C07257=1094.933,100.327,-61.473,176.140,17.129,152.422
C07258=1094.927,100.078,-61.455,176.137,17.128,152.422
C07259=1094.922,99.829,-61.436,176.135,17.127,152.422
C07260=1094.916,99.579,-61.418,176.132,17.127,152.423
C07261=1094.911,99.330,-61.401,176.130,17.125,152.423
C07262=1094.905,99.081,-61.381,176.128,17.125,152.423
C07263=1094.899,98.832,-61.364,176.125,17.124,152.424
C07264=1094.893,98.582,-61.346,176.123,17.123,152.424
C07265=1094.888,98.333,-61.327,176.120,17.123,152.424
C07266=1094.882,98.083,-61.309,176.117,17.121,152.425
C07267=1094.877,97.834,-61.291,176.115,17.121,152.425
C07268=1094.870,97.585,-61.274,176.112,17.120,152.425
C07269=1094.865,97.336,-61.255,176.110,17.119,152.426
C07270=1094.859,97.086,-61.237,176.108,17.118,152.426
C07271=1094.854,96.837,-61.219,176.106,17.117,152.426
C07272=1094.848,96.587,-61.201,176.103,17.117,152.426
C07273=1094.843,96.339,-61.182,176.100,17.115,152.427
C07274=1094.836,96.063,-61.163,176.098,17.115,152.427
C07275=1094.830,95.788,-61.143,176.095,17.114,152.427
C07276=1094.824,95.513,-61.123,176.093,17.113,152.428
C07277=1094.817,95.237,-61.104,176.090,17.112,152.428
C07278=1094.812,94.988,-61.085,176.087,17.111,152.428
C07279=1094.806,94.739,-61.067,176.085,17.110,152.429
C07280=1094.801,94.490,-61.049,176.082,17.109,152.429
C07281=1094.794,94.240,-61.031,176.080,17.108,152.429
C07282=1094.790,93.991,-61.013,176.077,17.108,152.430
C07283=1094.784,93.741,-60.995,176.075,17.107,152.430
C07284=1094.778,93.492,-60.978,176.073,17.106,152.430
C07285=1094.772,93.243,-60.960,176.070,17.104,152.430
C07286=1094.767,92.993,-60.941,176.068,17.104,152.431
C07287=1094.761,92.744,-60.923,176.065,17.103,152.431
C07288=1094.756,92.495,-60.906,176.063,17.102,152.431
C07289=1094.750,92.245,-60.888,176.061,17.101,152.432
C07290=1094.744,91.996,-60.870,176.059,17.101,152.432
C07291=1094.739,91.747,-60.852,176.056,17.099,152.432
C07292=1094.733,91.497,-60.834,176.054,17.099,152.432
C07293=1094.728,91.248,-60.816,176.051,17.097,152.433
C07294=1094.722,90.999,-60.799,176.048,17.097,152.433
C07295=1094.716,90.749,-60.781,176.046,17.096,152.433
C07296=1094.711,90.500,-60.763,176.044,17.095,152.434
C07297=1094.705,90.251,-60.746,176.042,17.094,152.434
C07298=1094.699,90.002,-60.728,176.039,17.093,152.434
C07299=1094.693,89.753,-60.710,176.037,17.093,152.434
C07300=1094.688,89.504,-60.693,176.034,17.092,152.435
C07301=1094.682,89.254,-60.675,176.032,17.091,152.435
C07302=1094.676,89.005,-60.657,176.030,17.090,152.435
C07303=1094.670,88.755,-60.639,176.027,17.088,152.436
C07304=1094.665,88.506,-60.622,176.025,17.088,152.436
C07305=1094.659,88.257,-60.604,176.022,17.087,152.436
C07306=1094.653,88.007,-60.586,176.020,17.086,152.436
C07307=1094.647,87.758,-60.569,176.017,17.085,152.437
C07308=1094.642,87.509,-60.551,176.015,17.084,152.437
C07309=1094.636,87.260,-60.534,176.013,17.083,152.437
C07310=1094.631,87.010,-60.516,176.011,17.083,152.437
C07311=1094.625,86.761,-60.499,176.008,17.081,152.438
C07312=1094.620,86.512,-60.481,176.006,17.081,152.438
C07313=1094.613,86.262,-60.463,176.004,17.079,152.438
C07314=1094.608,86.013,-60.446,176.001,17.078,152.439
C07315=1094.602,85.764,-60.428,175.999,17.078,152.439
C07316=1094.596,85.514,-60.410,175.996,17.076,152.439
C07317=1094.591,85.264,-60.393,175.994,17.076,152.439
C07318=1094.586,85.015,-60.376,175.992,17.074,152.440
C07319=1094.580,84.766,-60.358,175.990,17.074,152.440
C07320=1094.574,84.517,-60.340,175.987,17.073,152.440
C07321=1094.568,84.268,-60.323,175.985,17.072,152.440
C07322=1094.563,84.018,-60.306,175.982,17.071,152.441
C07323=1094.558,83.769,-60.288,175.981,17.070,152.441
C07324=1094.552,83.519,-60.270,175.978,17.069,152.441
C07325=1094.546,83.270,-60.253,175.976,17.068,152.441
C07326=1094.540,83.021,-60.237,175.973,17.067,152.442
C07327=1094.535,82.772,-60.219,175.970,17.066,152.442
C07328=1094.529,82.523,-60.201,175.969,17.065,152.442
C07329=1094.523,82.273,-60.183,175.966,17.064,152.442
C07330=1094.518,82.023,-60.167,175.964,17.063,152.443
C07331=1094.512,81.774,-60.149,175.961,17.062,152.443
C07332=1094.507,81.525,-60.131,175.959,17.061,152.443
C07333=1094.501,81.276,-60.115,175.957,17.060,152.443
C07334=1094.495,81.026,-60.097,175.955,17.059,152.444
C07335=1094.489,80.777,-60.080,175.952,17.058,152.444
C07336=1094.484,80.527,-60.063,175.950,17.058,152.444
C07337=1094.478,80.278,-60.045,175.947,17.056,152.445
C07338=1094.472,80.003,-60.026,175.945,17.055,152.445
C07339=1094.466,79.728,-60.007,175.943,17.054,152.445
C07340=1094.460,79.452,-59.988,175.940,17.053,152.445
C07341=1094.454,79.177,-59.969,175.937,17.052,152.446
C07342=1094.448,78.928,-59.951,175.935,17.050,152.446
C07343=1094.443,78.678,-59.934,175.933,17.050,152.446
C07344=1094.437,78.429,-59.918,175.930,17.048,152.446
C07345=1094.431,78.180,-59.900,175.928,17.048,152.447
C07346=1094.425,77.930,-59.883,175.926,17.047,152.447
C07347=1094.420,77.681,-59.865,175.924,17.046,152.447
C07348=1094.414,77.431,-59.849,175.921,17.045,152.447
C07349=1094.408,77.182,-59.831,175.919,17.044,152.448
C07350=1094.403,76.933,-59.814,175.917,17.043,152.448
C07351=1094.397,76.684,-59.798,175.915,17.042,152.448
C07352=1094.391,76.434,-59.780,175.912,17.040,152.448
C07353=1094.385,76.185,-59.763,175.910,17.040,152.448
C07354=1094.379,75.935,-59.746,175.908,17.039,152.449
C07355=1094.374,75.686,-59.729,175.906,17.038,152.449
C07356=1094.369,75.437,-59.712,175.903,17.037,152.449
C07357=1094.363,75.188,-59.695,175.901,17.036,152.450
C07358=1094.357,74.938,-59.678,175.899,17.034,152.450
C07359=1094.352,74.689,-59.661,175.897,17.034,152.450
C07360=1094.345,74.439,-59.644,175.894,17.033,152.450
C07361=1094.340,74.190,-59.626,175.892,17.032,152.450
C07362=1094.334,73.940,-59.610,175.889,17.031,152.451
C07363=1094.329,73.691,-59.593,175.888,17.030,152.451
C07364=1094.323,73.442,-59.576,175.885,17.028,152.451
C07365=1094.318,73.192,-59.559,175.883,17.028,152.451
C07366=1094.312,72.944,-59.542,175.880,17.026,152.452
C07367=1094.306,72.694,-59.525,175.879,17.026,152.452
C07368=1094.300,72.445,-59.509,175.876,17.024,152.452
C07369=1094.295,72.196,-59.491,175.874,17.023,152.452
C07370=1094.290,71.946,-59.474,175.872,17.022,152.452
C07371=1094.283,71.696,-59.458,175.870,17.022,152.453
C07372=1094.278,71.447,-59.440,175.867,17.020,152.453
C07373=1094.272,71.197,-59.424,175.865,17.019,152.453
C07374=1094.266,70.948,-59.407,175.863,17.018,152.453
C07375=1094.261,70.699,-59.390,175.861,17.017,152.453
C07376=1094.255,70.449,-59.373,175.858,17.016,152.454
C07377=1094.250,70.200,-59.356,175.856,17.015,152.454
C07378=1094.243,69.951,-59.340,175.854,17.014,152.454
C07379=1094.238,69.701,-59.323,175.852,17.013,152.454
C07380=1094.232,69.452,-59.306,175.849,17.011,152.455
C07381=1094.227,69.202,-59.290,175.847,17.011,152.455
C07382=1094.221,68.954,-59.273,175.845,17.010,152.455
C07383=1094.216,68.704,-59.256,175.843,17.008,152.455
C07384=1094.210,68.455,-59.239,175.840,17.007,152.456
C07385=1094.204,68.205,-59.223,175.838,17.007,152.456
C07386=1094.198,67.956,-59.206,175.836,17.005,152.456
C07387=1094.193,67.707,-59.189,175.834,17.004,152.456
C07388=1094.187,67.457,-59.173,175.831,17.003,152.456
C07389=1094.182,67.208,-59.156,175.830,17.002,152.457
C07390=1094.176,66.958,-59.139,175.827,17.001,152.457
C07391=1094.170,66.709,-59.123,175.825,17.000,152.457
C07392=1094.164,66.460,-59.106,175.824,16.999,152.457
C07393=1094.158,66.211,-59.089,175.821,16.998,152.457
C07394=1094.153,65.961,-59.072,175.819,16.997,152.458
C07395=1094.147,65.711,-59.056,175.817,16.995,152.458
C07396=1094.141,65.462,-59.040,175.815,16.995,152.458
C07397=1094.136,65.212,-59.023,175.812,16.993,152.458
C07398=1094.130,64.963,-59.007,175.810,16.992,152.458
C07399=1094.125,64.714,-58.989,175.808,16.991,152.459
C07400=1094.119,64.465,-58.973,175.806,16.990,152.459
C07401=1094.113,64.215,-58.957,175.803,16.989,152.459
C07402=1094.106,63.940,-58.939,175.801,16.988,152.459
C07403=1094.100,63.664,-58.921,175.799,16.987,152.460
C07404=1094.093,63.389,-58.903,175.796,16.986,152.460
C07405=1094.087,63.113,-58.885,175.794,16.984,152.460
C07406=1094.082,62.864,-58.867,175.792,16.983,152.460
C07407=1094.076,62.615,-58.851,175.789,16.982,152.461
C07408=1094.070,62.366,-58.835,175.787,16.981,152.461
C07409=1094.064,62.116,-58.818,175.785,16.980,152.461
C07410=1094.058,61.867,-58.802,175.783,16.979,152.461
C07411=1094.053,61.617,-58.785,175.781,16.978,152.461
C07412=1094.047,61.368,-58.769,175.778,16.977,152.462
C07413=1094.041,61.119,-58.753,175.777,16.976,152.462
C07414=1094.035,60.869,-58.736,175.774,16.974,152.462
C07415=1094.029,60.620,-58.720,175.772,16.974,152.462
C07416=1094.024,60.370,-58.703,175.770,16.972,152.462
C07417=1094.018,60.121,-58.687,175.768,16.971,152.463
C07418=1094.012,59.871,-58.672,175.765,16.970,152.463
C07419=1094.006,59.622,-58.655,175.763,16.969,152.463
C07420=1094.000,59.372,-58.639,175.762,16.968,152.463
C07421=1093.995,59.123,-58.622,175.759,16.967,152.463
C07422=1093.989,58.873,-58.606,175.757,16.966,152.464
C07423=1093.983,58.624,-58.590,175.755,16.964,152.464
C07424=1093.978,58.375,-58.574,175.753,16.964,152.464
C07425=1093.972,58.126,-58.558,175.750,16.962,152.464
C07426=1093.966,57.877,-58.541,175.749,16.961,152.464
C07427=1093.960,57.627,-58.525,175.746,16.960,152.464
C07428=1093.955,57.377,-58.509,175.744,16.959,152.465
C07429=1093.949,57.128,-58.493,175.742,16.958,152.465
C07430=1093.943,56.878,-58.476,175.740,16.957,152.465
C07431=1093.937,56.629,-58.460,175.738,16.956,152.465
C07432=1093.931,56.380,-58.444,175.736,16.954,152.465
C07433=1093.926,56.131,-58.428,175.734,16.954,152.466
C07434=1093.920,55.881,-58.412,175.731,16.952,152.466
C07435=1093.915,55.631,-58.396,175.729,16.951,152.466
C07436=1093.909,55.382,-58.379,175.727,16.949,152.466
C07437=1093.903,55.133,-58.363,175.725,16.949,152.466
C07438=1093.897,54.883,-58.347,175.723,16.947,152.467
C07439=1093.892,54.633,-58.331,175.721,16.946,152.467
C07440=1093.886,54.385,-58.315,175.719,16.945,152.467
C07441=1093.880,54.135,-58.299,175.717,16.944,152.467
C07442=1093.874,53.886,-58.283,175.715,16.943,152.467
C07443=1093.869,53.636,-58.267,175.712,16.941,152.467
C07444=1093.863,53.387,-58.251,175.710,16.941,152.468
C07445=1093.857,53.137,-58.234,175.708,16.939,152.468
C07446=1093.852,52.888,-58.219,175.706,16.938,152.468
C07447=1093.846,52.638,-58.203,175.704,16.937,152.468
C07448=1093.841,52.389,-58.187,175.702,16.935,152.468
C07449=1093.835,52.139,-58.171,175.700,16.935,152.468
C07450=1093.829,51.890,-58.155,175.698,16.933,152.469
C07451=1093.824,51.641,-58.139,175.696,16.932,152.469
C07452=1093.818,51.391,-58.123,175.693,16.931,152.469
C07453=1093.812,51.142,-58.107,175.692,16.930,152.469
C07454=1093.806,50.892,-58.091,175.690,16.929,152.469
C07455=1093.801,50.643,-58.076,175.687,16.927,152.469
C07456=1093.795,50.394,-58.059,175.686,16.926,152.470
C07457=1093.789,50.144,-58.043,175.683,16.925,152.470
C07458=1093.783,49.894,-58.028,175.681,16.924,152.470
C07459=1093.778,49.646,-58.012,175.679,16.922,152.470
C07460=1093.772,49.396,-57.996,175.677,16.921,152.470
C07461=1093.766,49.147,-57.980,175.676,16.920,152.470
C07462=1093.761,48.897,-57.964,175.673,16.919,152.471
C07463=1093.755,48.648,-57.948,175.671,16.918,152.471
C07464=1093.750,48.399,-57.932,175.669,16.916,152.471
C07465=1093.744,48.149,-57.917,175.667,16.915,152.471
C07466=1093.738,47.873,-57.899,175.664,16.914,152.471
C07467=1093.732,47.598,-57.882,175.663,16.913,152.471
C07468=1093.726,47.321,-57.864,175.660,16.911,152.472
C07469=1093.720,47.046,-57.846,175.658,16.910,152.472
C07470=1093.714,46.796,-57.831,175.656,16.909,152.472
C07471=1093.708,46.548,-57.815,175.654,16.907,152.472
C07472=1093.702,46.298,-57.800,175.652,16.906,152.472
C07473=1093.696,46.048,-57.784,175.649,16.905,152.472
C07474=1093.691,45.799,-57.769,175.648,16.904,152.472
C07475=1093.685,45.550,-57.752,175.646,16.902,152.473
C07476=1093.680,45.300,-57.737,175.643,16.901,152.473
C07477=1093.674,45.051,-57.721,175.642,16.900,152.473
C07478=1093.669,44.801,-57.705,175.639,16.898,152.473
C07479=1093.663,44.551,-57.690,175.638,16.897,152.473
C07480=1093.658,44.303,-57.674,175.636,16.897,152.473
C07481=1093.652,44.053,-57.658,175.633,16.895,152.474
C07482=1093.647,43.804,-57.642,175.632,16.894,152.474
C07483=1093.641,43.554,-57.627,175.629,16.892,152.474
C07484=1093.635,43.304,-57.611,175.627,16.891,152.474
C07485=1093.629,43.055,-57.596,175.626,16.890,152.474
C07486=1093.624,42.806,-57.580,175.623,16.889,152.474
C07487=1093.618,42.556,-57.565,175.622,16.887,152.474
C07488=1093.612,42.306,-57.549,175.619,16.886,152.475
C07489=1093.607,42.057,-57.534,175.617,16.885,152.475
C07490=1093.600,41.808,-57.518,175.616,16.884,152.475
C07491=1093.595,41.558,-57.502,175.613,16.882,152.475
C07492=1093.590,41.309,-57.487,175.611,16.882,152.475
C07493=1093.584,41.059,-57.472,175.609,16.880,152.475
C07494=1093.578,40.811,-57.456,175.607,16.879,152.475
C07495=1093.572,40.561,-57.441,175.606,16.878,152.476
C07496=1093.567,40.311,-57.425,175.603,16.876,152.476
C07497=1093.561,40.062,-57.409,175.601,16.875,152.476
C07498=1093.555,39.812,-57.394,175.599,16.874,152.476
C07499=1093.549,39.562,-57.379,175.597,16.872,152.476
C07500=1093.544,39.313,-57.364,175.596,16.871,152.476
C07501=1093.538,39.064,-57.347,175.593,16.870,152.477
C07502=1093.532,38.815,-57.333,175.591,16.869,152.477
C07503=1093.527,38.565,-57.317,175.589,16.867,152.477
C07504=1093.521,38.315,-57.302,175.587,16.866,152.477
C07505=1093.516,38.066,-57.286,175.586,16.865,152.477
C07506=1093.509,37.817,-57.271,175.583,16.864,152.477
C07507=1093.504,37.567,-57.256,175.582,16.863,152.477
C07508=1093.498,37.318,-57.241,175.580,16.861,152.477
C07509=1093.492,37.068,-57.225,175.577,16.860,152.478
C07510=1093.487,36.818,-57.210,175.576,16.859,152.478
C07511=1093.481,36.569,-57.194,175.573,16.857,152.478
C07512=1093.476,36.320,-57.179,175.572,16.856,152.478
C07513=1093.469,36.071,-57.164,175.570,16.855,152.478
C07514=1093.464,35.821,-57.149,175.567,16.853,152.478
C07515=1093.459,35.571,-57.134,175.566,16.853,152.479
C07516=1093.452,35.322,-57.119,175.564,16.852,152.479
C07517=1093.447,35.072,-57.103,175.562,16.850,152.479
C07518=1093.440,34.823,-57.088,175.560,16.849,152.479
C07519=1093.435,34.573,-57.072,175.557,16.847,152.479
C07520=1093.429,34.324,-57.058,175.556,16.847,152.479
C07521=1093.423,34.074,-57.042,175.554,16.845,152.479
C07522=1093.418,33.825,-57.028,175.552,16.844,152.479
C07523=1093.412,33.576,-57.012,175.550,16.843,152.480
C07524=1093.406,33.327,-56.997,175.548,16.841,152.480
C07525=1093.400,33.077,-56.982,175.546,16.840,152.480
C07526=1093.395,32.827,-56.966,175.544,16.839,152.480
C07527=1093.389,32.578,-56.952,175.542,16.838,152.480
C07528=1093.383,32.328,-56.936,175.540,16.836,152.480
C07529=1093.378,32.079,-56.922,175.538,16.835,152.480
C07530=1093.371,31.803,-56.905,175.536,16.833,152.480
C07531=1093.365,31.528,-56.888,175.534,16.832,152.481
C07532=1093.359,31.252,-56.871,175.532,16.831,152.481
C07533=1093.352,30.977,-56.855,175.529,16.829,152.481
C07534=1093.347,30.727,-56.839,175.527,16.828,152.481
C07535=1093.341,30.478,-56.825,175.526,16.827,152.481
C07536=1093.335,30.228,-56.809,175.523,16.825,152.481
C07537=1093.330,29.979,-56.795,175.522,16.824,152.481
C07538=1093.324,29.729,-56.779,175.520,16.823,152.482
C07539=1093.318,29.480,-56.765,175.518,16.821,152.482
C07540=1093.312,29.230,-56.749,175.516,16.820,152.482
C07541=1093.307,28.981,-56.734,175.515,16.819,152.482
C07542=1093.301,28.731,-56.720,175.512,16.817,152.482
C07543=1093.296,28.481,-56.705,175.511,16.816,152.482
C07544=1093.289,28.232,-56.690,175.508,16.815,152.482
C07545=1093.284,27.983,-56.675,175.506,16.814,152.482
C07546=1093.278,27.733,-56.660,175.505,16.813,152.483
C07547=1093.272,27.484,-56.645,175.502,16.811,152.483
C07548=1093.266,27.234,-56.630,175.501,16.810,152.483
C07549=1093.261,26.985,-56.615,175.499,16.809,152.483
C07550=1093.254,26.735,-56.601,175.496,16.807,152.483
C07551=1093.249,26.485,-56.586,175.495,16.806,152.483
C07552=1093.244,26.236,-56.571,175.493,16.805,152.483
C07553=1093.237,25.987,-56.556,175.491,16.803,152.483
C07554=1093.232,25.738,-56.541,175.489,16.802,152.483
C07555=1093.226,25.488,-56.526,175.487,16.801,152.484
C07556=1093.220,25.238,-56.512,175.485,16.800,152.484
C07557=1093.215,24.988,-56.497,175.483,16.799,152.484
C07558=1093.209,24.739,-56.482,175.482,16.797,152.484
C07559=1093.203,24.490,-56.467,175.479,16.796,152.484
C07560=1093.197,24.240,-56.452,175.478,16.795,152.484
C07561=1093.191,23.990,-56.438,175.476,16.793,152.484
C07562=1093.186,23.741,-56.423,175.474,16.792,152.485
C07563=1093.180,23.492,-56.409,175.472,16.791,152.485
C07564=1093.174,23.242,-56.393,175.470,16.789,152.485
C07565=1093.169,22.993,-56.379,175.468,16.788,152.485
C07566=1093.162,22.743,-56.364,175.466,16.787,152.485
C07567=1093.157,22.494,-56.349,175.465,16.786,152.485
C07568=1093.152,22.244,-56.335,175.462,16.784,152.485
C07569=1093.145,21.995,-56.320,175.461,16.783,152.485
C07570=1093.140,21.746,-56.306,175.459,16.782,152.485
C07571=1093.134,21.495,-56.291,175.457,16.780,152.485
C07572=1093.129,21.246,-56.276,175.455,16.779,152.486
C07573=1093.123,20.997,-56.262,175.453,16.778,152.486
C07574=1093.117,20.747,-56.248,175.451,16.776,152.486
C07575=1093.112,20.498,-56.232,175.449,16.775,152.486
C07576=1093.105,20.248,-56.217,175.448,16.774,152.486
C07577=1093.100,19.998,-56.204,175.446,16.772,152.486
C07578=1093.094,19.749,-56.189,175.444,16.771,152.486
C07579=1093.088,19.500,-56.174,175.442,16.770,152.486
C07580=1093.082,19.250,-56.160,175.440,16.769,152.486
C07581=1093.077,19.001,-56.145,175.438,16.767,152.487
C07582=1093.071,18.751,-56.131,175.436,16.766,152.487
C07583=1093.065,18.502,-56.116,175.435,16.765,152.487
C07584=1093.059,18.252,-56.101,175.432,16.763,152.487
C07585=1093.053,18.002,-56.087,175.430,16.762,152.487
C07586=1093.048,17.753,-56.073,175.429,16.761,152.487
C07587=1093.042,17.503,-56.059,175.427,16.759,152.487
C07588=1093.036,17.254,-56.043,175.425,16.758,152.487
C07589=1093.031,17.004,-56.030,175.423,16.757,152.487
C07590=1093.025,16.755,-56.015,175.422,16.755,152.488
C07591=1093.019,16.505,-56.001,175.419,16.754,152.488
C07592=1093.013,16.256,-55.986,175.418,16.753,152.488
C07593=1093.007,16.006,-55.972,175.416,16.751,152.488
C07594=1093.001,15.733,-55.956,175.414,16.750,152.488
C07595=1092.995,15.458,-55.940,175.412,16.749,152.488
C07596=1092.988,15.184,-55.924,175.410,16.747,152.488
C07597=1092.982,14.909,-55.909,175.407,16.745,152.488
C07598=1092.976,14.660,-55.894,175.406,16.744,152.488
C07599=1092.971,14.410,-55.880,175.404,16.743,152.489
C07600=1092.965,14.162,-55.865,175.402,16.742,152.489
C07601=1092.959,13.912,-55.851,175.400,16.740,152.489
C07602=1092.953,13.663,-55.837,175.398,16.739,152.489
C07603=1092.947,13.412,-55.823,175.397,16.738,152.489
C07604=1092.941,13.163,-55.809,175.394,16.736,152.489
C07605=1092.936,12.914,-55.794,175.393,16.735,152.489
C07606=1092.929,12.663,-55.780,175.391,16.734,152.489
C07607=1092.924,12.415,-55.765,175.389,16.733,152.489
C07608=1092.918,12.165,-55.752,175.387,16.731,152.490
C07609=1092.913,11.915,-55.738,175.385,16.730,152.490
C07610=1092.906,11.666,-55.723,175.384,16.729,152.490
C07611=1092.901,11.416,-55.709,175.381,16.727,152.490
C07612=1092.895,11.167,-55.694,175.380,16.726,152.490
C07613=1092.889,10.917,-55.680,175.378,16.725,152.490
C07614=1092.883,10.668,-55.667,175.376,16.724,152.490
C07615=1092.877,10.419,-55.652,175.374,16.722,152.490
C07616=1092.871,10.168,-55.638,175.372,16.721,152.490
C07617=1092.865,9.919,-55.624,175.371,16.720,152.491
C07618=1092.860,9.670,-55.609,175.368,16.718,152.491
C07619=1092.854,9.420,-55.596,175.367,16.717,152.491
C07620=1092.848,9.170,-55.581,175.365,16.716,152.491
C07621=1092.842,8.921,-55.567,175.364,16.715,152.491
C07622=1092.836,8.672,-55.554,175.361,16.713,152.491
C07623=1092.831,8.422,-55.540,175.360,16.712,152.491
C07624=1092.825,8.172,-55.525,175.358,16.711,152.491
C07625=1092.819,7.923,-55.511,175.356,16.710,152.491
C07626=1092.813,7.673,-55.497,175.354,16.708,152.492
C07627=1092.808,7.424,-55.483,175.352,16.707,152.492
C07628=1092.802,7.174,-55.469,175.351,16.705,152.492
C07629=1092.796,6.925,-55.454,175.348,16.703,152.492
C07630=1092.790,6.675,-55.441,175.347,16.702,152.492
C07631=1092.784,6.426,-55.427,175.345,16.701,152.492
C07632=1092.778,6.176,-55.413,175.344,16.700,152.492
C07633=1092.773,5.926,-55.399,175.341,16.698,152.492
C07634=1092.767,5.677,-55.385,175.340,16.697,152.492
C07635=1092.761,5.427,-55.371,175.338,16.696,152.492
C07636=1092.755,5.178,-55.357,175.336,16.695,152.492
C07637=1092.749,4.928,-55.343,175.334,16.693,152.493
C07638=1092.744,4.678,-55.329,175.332,16.692,152.493
C07639=1092.738,4.429,-55.315,175.331,16.691,152.493
C07640=1092.732,4.180,-55.301,175.329,16.689,152.493
C07641=1092.726,3.931,-55.288,175.327,16.688,152.493
C07642=1092.721,3.681,-55.274,175.325,16.686,152.493
C07643=1092.715,3.431,-55.259,175.324,16.685,152.493
C07644=1092.709,3.181,-55.246,175.322,16.684,152.493
C07645=1092.704,2.931,-55.232,175.320,16.682,152.493
C07646=1092.697,2.682,-55.218,175.318,16.681,152.493
C07647=1092.692,2.433,-55.205,175.316,16.680,152.493
C07648=1092.686,2.184,-55.190,175.315,16.679,152.493
C07649=1092.681,1.934,-55.176,175.313,16.677,152.494
C07650=1092.675,1.684,-55.162,175.311,16.676,152.494
C07651=1092.668,1.435,-55.149,175.309,16.675,152.494
C07652=1092.663,1.185,-55.135,175.308,16.673,152.494
C07653=1092.658,0.935,-55.121,175.305,16.672,152.494
C07654=1092.652,0.686,-55.107,175.304,16.671,152.494
C07655=1092.646,0.437,-55.094,175.302,16.669,152.494
C07656=1092.640,0.187,-55.080,175.301,16.668,152.494
C07657=1092.635,-0.063,-55.066,175.298,16.666,152.494
C07658=1092.628,-0.335,-55.051,175.297,16.665,152.494
C07659=1092.622,-0.607,-55.036,175.294,16.663,152.495
C07660=1092.616,-0.880,-55.021,175.293,16.662,152.495
C07661=1092.610,-1.152,-55.006,175.291,16.660,152.495
C07662=1092.604,-1.401,-54.992,175.289,16.659,152.495
C07663=1092.598,-1.650,-54.979,175.287,16.658,152.495
C07664=1092.593,-1.900,-54.965,175.286,16.657,152.495
C07665=1092.587,-2.150,-54.951,175.283,16.655,152.495
C07666=1092.581,-2.400,-54.938,175.282,16.654,152.495
C07667=1092.575,-2.649,-54.924,175.280,16.652,152.495
C07668=1092.570,-2.899,-54.910,175.279,16.651,152.495
C07669=1092.564,-3.148,-54.896,175.277,16.650,152.495
C07670=1092.558,-3.398,-54.883,175.275,16.648,152.495
C07671=1092.552,-3.647,-54.869,175.273,16.647,152.496
C07672=1092.546,-3.896,-54.856,175.272,16.646,152.496
C07673=1092.541,-4.146,-54.842,175.270,16.645,152.496
C07674=1092.535,-4.396,-54.829,175.267,16.643,152.496
C07675=1092.529,-4.645,-54.816,175.266,16.641,152.496
C07676=1092.523,-4.895,-54.802,175.265,16.640,152.496
C07677=1092.518,-5.144,-54.788,175.263,16.639,152.496
C07678=1092.511,-5.394,-54.775,175.261,16.638,152.496
C07679=1092.505,-5.644,-54.761,175.259,16.636,152.496
C07680=1092.499,-5.893,-54.748,175.257,16.635,152.496
C07681=1092.494,-6.143,-54.735,175.256,16.634,152.496
C07682=1092.488,-6.393,-54.721,175.254,16.633,152.497
C07683=1092.482,-6.642,-54.707,175.252,16.631,152.497
C07684=1092.476,-6.891,-54.694,175.250,16.630,152.497
C07685=1092.471,-7.141,-54.680,175.249,16.628,152.497
C07686=1092.464,-7.390,-54.667,175.247,16.627,152.497
C07687=1092.459,-7.640,-54.654,175.245,16.626,152.497
C07688=1092.453,-7.890,-54.641,175.243,16.624,152.497
C07689=1092.447,-8.139,-54.627,175.241,16.623,152.497
C07690=1092.441,-8.389,-54.613,175.240,16.622,152.497
C07691=1092.436,-8.639,-54.600,175.238,16.621,152.497
C07692=1092.430,-8.888,-54.587,175.236,16.619,152.497
C07693=1092.424,-9.137,-54.574,175.234,16.618,152.497
C07694=1092.418,-9.387,-54.560,175.233,16.617,152.498
C07695=1092.412,-9.637,-54.547,175.231,16.615,152.498
C07696=1092.407,-9.886,-54.533,175.230,16.614,152.498
C07697=1092.400,-10.136,-54.520,175.227,16.613,152.498
C07698=1092.395,-10.386,-54.506,175.226,16.611,152.498
C07699=1092.389,-10.636,-54.493,175.224,16.610,152.498
C07700=1092.383,-10.885,-54.480,175.223,16.609,152.498
C07701=1092.378,-11.134,-54.467,175.221,16.608,152.498
C07702=1092.372,-11.384,-54.454,175.219,16.606,152.498
C07703=1092.366,-11.633,-54.440,175.217,16.605,152.498
C07704=1092.360,-11.883,-54.427,175.215,16.604,152.499
C07705=1092.355,-12.133,-54.414,175.214,16.602,152.498
C07706=1092.349,-12.382,-54.401,175.212,16.601,152.499
C07707=1092.342,-12.631,-54.387,175.210,16.599,152.499
C07708=1092.337,-12.881,-54.374,175.208,16.598,152.499
C07709=1092.331,-13.131,-54.361,175.207,16.597,152.499
C07710=1092.325,-13.380,-54.347,175.205,16.596,152.499
C07711=1092.320,-13.630,-54.334,175.204,16.594,152.499
C07712=1092.313,-13.879,-54.321,175.201,16.592,152.499
C07713=1092.308,-14.130,-54.308,175.200,16.591,152.499
C07714=1092.302,-14.379,-54.295,175.198,16.590,152.499
C07715=1092.296,-14.629,-54.281,175.196,16.589,152.499
C07716=1092.291,-14.878,-54.268,175.195,16.587,152.499
C07717=1092.284,-15.128,-54.255,175.194,16.586,152.499
C07718=1092.279,-15.378,-54.242,175.191,16.585,152.500
C07719=1092.273,-15.627,-54.229,175.189,16.583,152.500
C07720=1092.267,-15.877,-54.216,175.188,16.582,152.500
C07721=1092.261,-16.126,-54.203,175.186,16.581,152.500
C07722=1092.255,-16.397,-54.189,175.184,16.579,152.500
C07723=1092.249,-16.667,-54.174,175.182,16.578,152.500
C07724=1092.243,-16.938,-54.160,175.181,16.577,152.500
C07725=1092.236,-17.209,-54.146,175.178,16.575,152.500
C07726=1092.230,-17.458,-54.133,175.177,16.574,152.500
C07727=1092.224,-17.708,-54.120,175.175,16.573,152.500
C07728=1092.218,-17.957,-54.107,175.174,16.572,152.501
C07729=1092.212,-18.207,-54.094,175.172,16.570,152.501
C07730=1092.206,-18.456,-54.081,175.170,16.569,152.501
C07731=1092.201,-18.706,-54.069,175.168,16.567,152.501
C07732=1092.195,-18.955,-54.055,175.167,16.566,152.501
C07733=1092.189,-19.205,-54.043,175.165,16.565,152.501
C07734=1092.183,-19.454,-54.029,175.163,16.564,152.501
C07735=1092.177,-19.704,-54.016,175.162,16.563,152.501
C07736=1092.172,-19.954,-54.004,175.159,16.561,152.501
C07737=1092.165,-20.203,-53.990,175.158,16.560,152.501
C07738=1092.159,-20.453,-53.978,175.156,16.558,152.501
C07739=1092.153,-20.703,-53.965,175.155,16.557,152.501
C07740=1092.148,-20.953,-53.952,175.153,16.556,152.502
C07741=1092.142,-21.201,-53.939,175.152,16.555,152.502
C07742=1092.137,-21.451,-53.926,175.150,16.554,152.502
C07743=1092.131,-21.701,-53.913,175.148,16.552,152.502
C07744=1092.124,-21.950,-53.900,175.146,16.551,152.502
C07745=1092.118,-22.200,-53.888,175.145,16.549,152.502
C07746=1092.113,-22.450,-53.875,175.143,16.548,152.502
C07747=1092.107,-22.700,-53.861,175.141,16.547,152.502
C07748=1092.102,-22.949,-53.849,175.140,16.546,152.502
C07749=1092.096,-23.199,-53.837,175.137,16.544,152.502
C07750=1092.090,-23.448,-53.823,175.136,16.543,152.502
C07751=1092.084,-23.698,-53.811,175.134,16.541,152.502
C07752=1092.078,-23.948,-53.798,175.133,16.540,152.503
C07753=1092.072,-24.197,-53.785,175.131,16.539,152.503
C07754=1092.066,-24.446,-53.773,175.130,16.538,152.503
C07755=1092.061,-24.696,-53.760,175.128,16.537,152.503
C07756=1092.055,-24.946,-53.746,175.126,16.535,152.503
C07757=1092.049,-25.196,-53.734,175.124,16.533,152.503
C07758=1092.043,-25.445,-53.721,175.123,16.532,152.503
C07759=1092.037,-25.695,-53.709,175.121,16.531,152.503
C07760=1092.032,-25.944,-53.696,175.119,16.530,152.503
C07761=1092.026,-26.194,-53.683,175.118,16.529,152.503
C07762=1092.020,-26.444,-53.671,175.115,16.527,152.503
C07763=1092.014,-26.694,-53.658,175.114,16.525,152.503
C07764=1092.008,-26.942,-53.645,175.112,16.524,152.504
C07765=1092.002,-27.192,-53.633,175.111,16.523,152.504
C07766=1091.996,-27.442,-53.620,175.109,16.522,152.504
C07767=1091.991,-27.692,-53.607,175.108,16.521,152.504
C07768=1091.984,-27.941,-53.594,175.106,16.520,152.504
C07769=1091.978,-28.191,-53.582,175.104,16.519,152.504
C07770=1091.973,-28.440,-53.569,175.102,16.517,152.504
C07771=1091.967,-28.690,-53.557,175.101,16.515,152.504
C07772=1091.961,-28.940,-53.544,175.099,16.514,152.504
C07773=1091.955,-29.190,-53.532,175.097,16.513,152.504
C07774=1091.949,-29.439,-53.519,175.096,16.512,152.504
C07775=1091.943,-29.689,-53.506,175.094,16.511,152.505
C07776=1091.938,-29.938,-53.494,175.092,16.510,152.505
C07777=1091.931,-30.188,-53.482,175.091,16.508,152.505
C07778=1091.925,-30.438,-53.469,175.088,16.507,152.505
C07779=1091.919,-30.687,-53.457,175.087,16.505,152.505
C07780=1091.914,-30.937,-53.445,175.085,16.504,152.505
C07781=1091.908,-31.186,-53.431,175.084,16.503,152.505
C07782=1091.902,-31.436,-53.419,175.082,16.502,152.505
C07783=1091.896,-31.686,-53.406,175.081,16.501,152.505
C07784=1091.890,-31.935,-53.394,175.079,16.499,152.505
C07785=1091.885,-32.185,-53.381,175.077,16.498,152.505
C07786=1091.878,-32.455,-53.368,175.075,16.497,152.506
C07787=1091.872,-32.724,-53.354,175.074,16.495,152.506
C07788=1091.866,-32.994,-53.341,175.072,16.494,152.506
C07789=1091.859,-33.264,-53.328,175.070,16.493,152.506
C07790=1091.853,-33.513,-53.316,175.068,16.491,152.506
C07791=1091.847,-33.763,-53.303,175.066,16.490,152.506
C07792=1091.842,-34.013,-53.291,175.065,16.489,152.506
C07793=1091.836,-34.262,-53.278,175.063,16.488,152.506
C07794=1091.830,-34.512,-53.266,175.062,16.487,152.506
C07795=1091.825,-34.761,-53.254,175.060,16.485,152.506
C07796=1091.818,-35.010,-53.241,175.059,16.484,152.506
C07797=1091.812,-35.260,-53.228,175.057,16.483,152.506
C07798=1091.806,-35.511,-53.217,175.055,16.481,152.507
C07799=1091.801,-35.760,-53.204,175.053,16.480,152.507
C07800=1091.795,-36.010,-53.192,175.051,16.479,152.507
C07801=1091.789,-36.260,-53.179,175.050,16.477,152.507
C07802=1091.783,-36.509,-53.168,175.048,16.476,152.507
C07803=1091.777,-36.759,-53.155,175.047,16.475,152.507
C07804=1091.771,-37.008,-53.143,175.045,16.474,152.507
C07805=1091.766,-37.258,-53.130,175.044,16.472,152.507
C07806=1091.760,-37.507,-53.118,175.042,16.471,152.507
C07807=1091.754,-37.757,-53.105,175.040,16.470,152.507
C07808=1091.748,-38.006,-53.094,175.039,16.469,152.507
C07809=1091.742,-38.256,-53.081,175.037,16.468,152.508
C07810=1091.736,-38.506,-53.069,175.035,16.466,152.508
C07811=1091.731,-38.755,-53.056,175.033,16.465,152.508
C07812=1091.724,-39.005,-53.045,175.032,16.463,152.508
C07813=1091.718,-39.255,-53.032,175.030,16.462,152.508
C07814=1091.713,-39.504,-53.020,175.029,16.461,152.508
C07815=1091.707,-39.754,-53.009,175.027,16.460,152.508
C07816=1091.701,-40.004,-52.996,175.025,16.459,152.508
C07817=1091.695,-40.253,-52.984,175.024,16.458,152.508
C07818=1091.689,-40.503,-52.972,175.022,16.457,152.508
C07819=1091.683,-40.753,-52.959,175.020,16.456,152.508
C07820=1091.677,-41.002,-52.947,175.019,16.454,152.509
C07821=1091.671,-41.252,-52.936,175.017,16.453,152.509
C07822=1091.665,-41.502,-52.923,175.016,16.452,152.509
C07823=1091.659,-41.751,-52.911,175.013,16.450,152.509
C07824=1091.653,-42.001,-52.899,175.012,16.449,152.509
C07825=1091.648,-42.250,-52.887,175.010,16.448,152.509
C07826=1091.641,-42.499,-52.875,175.009,16.446,152.509
C07827=1091.636,-42.750,-52.863,175.007,16.445,152.509
C07828=1091.629,-42.999,-52.851,175.005,16.444,152.509
C07829=1091.624,-43.249,-52.839,175.004,16.443,152.509
C07830=1091.618,-43.498,-52.826,175.002,16.442,152.510
C07831=1091.612,-43.749,-52.815,175.001,16.441,152.510
C07832=1091.606,-43.998,-52.803,174.999,16.440,152.510
C07833=1091.600,-44.247,-52.791,174.997,16.439,152.510
C07834=1091.594,-44.497,-52.779,174.996,16.437,152.510
C07835=1091.589,-44.747,-52.767,174.994,16.436,152.510
C07836=1091.582,-44.997,-52.755,174.992,16.435,152.510
C07837=1091.577,-45.246,-52.743,174.991,16.434,152.510
C07838=1091.570,-45.495,-52.731,174.990,16.432,152.510
C07839=1091.565,-45.746,-52.719,174.988,16.431,152.510
C07840=1091.559,-45.995,-52.707,174.985,16.430,152.510
C07841=1091.553,-46.245,-52.695,174.984,16.428,152.511
C07842=1091.548,-46.494,-52.683,174.982,16.427,152.511
C07843=1091.541,-46.744,-52.672,174.981,16.426,152.511
C07844=1091.536,-46.993,-52.659,174.979,16.425,152.511
C07845=1091.529,-47.243,-52.648,174.977,16.424,152.511
C07846=1091.523,-47.493,-52.636,174.976,16.423,152.511
C07847=1091.517,-47.742,-52.624,174.974,16.422,152.511
C07848=1091.512,-47.993,-52.612,174.973,16.420,152.511
C07849=1091.506,-48.242,-52.600,174.971,16.419,152.511
C07850=1091.500,-48.512,-52.587,174.969,16.418,152.511
C07851=1091.493,-48.782,-52.575,174.968,16.417,152.512
C07852=1091.487,-49.052,-52.562,174.966,16.415,152.512
C07853=1091.480,-49.322,-52.549,174.964,16.414,152.512
C07854=1091.475,-49.572,-52.537,174.962,16.413,152.512
C07855=1091.469,-49.821,-52.525,174.961,16.411,152.512
C07856=1091.463,-50.071,-52.513,174.959,16.410,152.512
C07857=1091.457,-50.320,-52.502,174.958,16.409,152.512
C07858=1091.451,-50.570,-52.489,174.956,16.408,152.512
C07859=1091.445,-50.820,-52.479,174.954,16.407,152.512
C07860=1091.439,-51.070,-52.466,174.953,16.406,152.512
C07861=1091.433,-51.320,-52.455,174.951,16.405,152.513
C07862=1091.427,-51.569,-52.443,174.949,16.404,152.513
C07863=1091.420,-51.818,-52.431,174.948,16.402,152.513
C07864=1091.415,-52.068,-52.420,174.946,16.401,152.513
C07865=1091.409,-52.318,-52.408,174.945,16.400,152.513
C07866=1091.402,-52.568,-52.397,174.943,16.399,152.513
C07867=1091.397,-52.817,-52.384,174.941,16.398,152.513
C07868=1091.391,-53.067,-52.373,174.940,16.397,152.513
C07869=1091.385,-53.316,-52.361,174.938,16.396,152.514
C07870=1091.378,-53.566,-52.350,174.936,16.395,152.514
C07871=1091.373,-53.816,-52.338,174.935,16.394,152.514
C07872=1091.367,-54.066,-52.327,174.933,16.393,152.514
C07873=1091.360,-54.315,-52.315,174.931,16.392,152.514
C07874=1091.355,-54.565,-52.303,174.930,16.390,152.514
C07875=1091.348,-54.815,-52.291,174.928,16.389,152.514
C07876=1091.343,-55.064,-52.281,174.927,16.388,152.514
C07877=1091.336,-55.314,-52.269,174.925,16.387,152.514
C07878=1091.331,-55.564,-52.257,174.923,16.386,152.514
C07879=1091.324,-55.813,-52.245,174.922,16.385,152.515
C07880=1091.319,-56.063,-52.234,174.920,16.384,152.515
C07881=1091.312,-56.313,-52.223,174.918,16.382,152.515
C07882=1091.307,-56.562,-52.211,174.917,16.381,152.515
C07883=1091.301,-56.812,-52.200,174.915,16.380,152.515
C07884=1091.295,-57.061,-52.188,174.914,16.379,152.515
C07885=1091.288,-57.311,-52.177,174.912,16.378,152.515
C07886=1091.282,-57.560,-52.165,174.910,16.377,152.515
C07887=1091.277,-57.811,-52.153,174.909,16.376,152.515
C07888=1091.271,-58.060,-52.142,174.907,16.375,152.516
C07889=1091.264,-58.310,-52.130,174.905,16.374,152.516
C07890=1091.259,-58.559,-52.120,174.904,16.373,152.516
C07891=1091.253,-58.810,-52.108,174.902,16.372,152.516
C07892=1091.247,-59.058,-52.096,174.900,16.370,152.516
C07893=1091.241,-59.309,-52.085,174.899,16.369,152.516
C07894=1091.235,-59.558,-52.073,174.897,16.368,152.516
C07895=1091.228,-59.808,-52.062,174.896,16.367,152.516
C07896=1091.223,-60.058,-52.051,174.894,16.366,152.517
C07897=1091.217,-60.307,-52.039,174.892,16.365,152.517
C07898=1091.211,-60.557,-52.028,174.891,16.364,152.517
C07899=1091.204,-60.807,-52.017,174.889,16.363,152.517
C07900=1091.198,-61.056,-52.005,174.888,16.361,152.517
C07901=1091.193,-61.305,-51.994,174.886,16.360,152.517
C07902=1091.187,-61.556,-51.982,174.884,16.359,152.517
C07903=1091.181,-61.805,-51.971,174.883,16.358,152.517
C07904=1091.175,-62.055,-51.959,174.881,16.357,152.517
C07905=1091.169,-62.304,-51.949,174.879,16.356,152.518
C07906=1091.163,-62.554,-51.937,174.878,16.355,152.518
C07907=1091.157,-62.804,-51.926,174.876,16.354,152.518
C07908=1091.152,-63.053,-51.914,174.874,16.353,152.518
C07909=1091.145,-63.303,-51.903,174.873,16.352,152.518
C07910=1091.139,-63.553,-51.892,174.872,16.351,152.518
C07911=1091.133,-63.803,-51.881,174.870,16.350,152.518
C07912=1091.127,-64.052,-51.869,174.869,16.349,152.518
C07913=1091.121,-64.301,-51.858,174.867,16.348,152.518
C07914=1091.115,-64.574,-51.846,174.865,16.347,152.519
C07915=1091.109,-64.844,-51.833,174.863,16.345,152.519
C07916=1091.102,-65.116,-51.822,174.861,16.344,152.519
C07917=1091.096,-65.387,-51.809,174.860,16.343,152.519
C07918=1091.089,-65.637,-51.798,174.858,16.342,152.519
C07919=1091.084,-65.886,-51.787,174.856,16.341,152.519
C07920=1091.078,-66.136,-51.776,174.855,16.340,152.519
C07921=1091.072,-66.386,-51.764,174.853,16.339,152.519
C07922=1091.066,-66.635,-51.753,174.851,16.337,152.520
C07923=1091.060,-66.885,-51.742,174.851,16.337,152.520
C07924=1091.054,-67.135,-51.731,174.849,16.336,152.520
C07925=1091.048,-67.384,-51.720,174.847,16.335,152.520
C07926=1091.043,-67.634,-51.709,174.846,16.334,152.520
C07927=1091.036,-67.884,-51.698,174.844,16.332,152.520
C07928=1091.031,-68.134,-51.687,174.843,16.331,152.520
C07929=1091.025,-68.383,-51.676,174.841,16.330,152.520
C07930=1091.019,-68.633,-51.663,174.839,16.329,152.521
C07931=1091.013,-68.883,-51.652,174.837,16.328,152.521
C07932=1091.007,-69.132,-51.642,174.836,16.327,152.521
C07933=1091.001,-69.382,-51.630,174.834,16.326,152.521
C07934=1090.995,-69.632,-51.619,174.833,16.325,152.521
C07935=1090.990,-69.881,-51.609,174.831,16.324,152.521
C07936=1090.983,-70.131,-51.597,174.829,16.323,152.521
C07937=1090.978,-70.381,-51.586,174.828,16.322,152.521
C07938=1090.972,-70.630,-51.576,174.826,16.320,152.521
C07939=1090.966,-70.880,-51.565,174.825,16.320,152.521
C07940=1090.960,-71.130,-51.553,174.823,16.319,152.522
C07941=1090.954,-71.380,-51.543,174.822,16.318,152.522
C07942=1090.948,-71.629,-51.532,174.820,16.317,152.522
C07943=1090.942,-71.879,-51.520,174.819,16.316,152.522
C07944=1090.936,-72.129,-51.510,174.817,16.315,152.522
C07945=1090.931,-72.378,-51.498,174.815,16.314,152.522
C07946=1090.925,-72.628,-51.487,174.814,16.312,152.522
C07947=1090.919,-72.878,-51.476,174.812,16.311,152.522
C07948=1090.913,-73.128,-51.465,174.810,16.311,152.523
C07949=1090.908,-73.377,-51.454,174.809,16.310,152.523
C07950=1090.902,-73.627,-51.443,174.807,16.308,152.523
C07951=1090.896,-73.877,-51.432,174.806,16.308,152.523
C07952=1090.890,-74.126,-51.421,174.805,16.307,152.523
C07953=1090.884,-74.376,-51.410,174.803,16.306,152.523
C07954=1090.878,-74.625,-51.400,174.801,16.304,152.523
C07955=1090.871,-74.875,-51.389,174.799,16.304,152.524
C07956=1090.865,-75.125,-51.378,174.798,16.303,152.524
C07957=1090.860,-75.374,-51.367,174.796,16.302,152.524
C07958=1090.853,-75.624,-51.356,174.795,16.300,152.524
C07959=1090.848,-75.874,-51.345,174.793,16.299,152.524
C07960=1090.842,-76.123,-51.334,174.791,16.299,152.524
C07961=1090.835,-76.373,-51.324,174.790,16.298,152.524
C07962=1090.829,-76.623,-51.313,174.789,16.297,152.524
C07963=1090.824,-76.873,-51.302,174.787,16.296,152.525
C07964=1090.818,-77.122,-51.292,174.785,16.295,152.525
C07965=1090.812,-77.373,-51.280,174.783,16.294,152.525
C07966=1090.806,-77.622,-51.269,174.782,16.293,152.525
C07967=1090.799,-77.871,-51.259,174.780,16.292,152.525
C07968=1090.794,-78.121,-51.248,174.779,16.291,152.525
C07969=1090.787,-78.371,-51.237,174.777,16.290,152.526
C07970=1090.782,-78.621,-51.227,174.776,16.289,152.526
C07971=1090.776,-78.870,-51.216,174.774,16.288,152.526
C07972=1090.770,-79.120,-51.205,174.773,16.287,152.526
C07973=1090.764,-79.369,-51.195,174.771,16.287,152.526
C07974=1090.758,-79.619,-51.184,174.769,16.285,152.526
C07975=1090.752,-79.869,-51.173,174.768,16.284,152.526
C07976=1090.746,-80.119,-51.163,174.766,16.283,152.526
C07977=1090.740,-80.368,-51.152,174.765,16.283,152.527
C07978=1090.734,-80.642,-51.140,174.762,16.281,152.527
C07979=1090.727,-80.915,-51.128,174.761,16.280,152.527
C07980=1090.721,-81.189,-51.117,174.759,16.280,152.527
C07981=1090.714,-81.463,-51.105,174.757,16.278,152.527
C07982=1090.707,-81.713,-51.094,174.756,16.277,152.527
C07983=1090.701,-81.962,-51.084,174.755,16.277,152.528
C07984=1090.695,-82.211,-51.073,174.753,16.276,152.528
C07985=1090.689,-82.461,-51.063,174.751,16.275,152.528
C07986=1090.682,-82.711,-51.052,174.749,16.274,152.528
C07987=1090.677,-82.961,-51.041,174.748,16.273,152.528
C07988=1090.670,-83.210,-51.031,174.746,16.272,152.528
C07989=1090.665,-83.460,-51.021,174.745,16.272,152.528
C07990=1090.658,-83.710,-51.009,174.743,16.271,152.529
C07991=1090.652,-83.960,-50.999,174.742,16.270,152.529
C07992=1090.647,-84.210,-50.989,174.740,16.269,152.529
C07993=1090.640,-84.459,-50.979,174.738,16.268,152.529
C07994=1090.634,-84.708,-50.968,174.736,16.267,152.529
C07995=1090.628,-84.958,-50.957,174.735,16.266,152.529
C07996=1090.622,-85.208,-50.947,174.734,16.266,152.529
C07997=1090.616,-85.458,-50.936,174.732,16.265,152.530
C07998=1090.610,-85.707,-50.926,174.730,16.264,152.530
C07999=1090.604,-85.957,-50.916,174.729,16.263,152.530
C08000=1090.598,-86.207,-50.904,174.727,16.262,152.530
C08001=1090.591,-86.456,-50.894,174.725,16.261,152.530
C08002=1090.586,-86.707,-50.884,174.725,16.260,152.530
C08003=1090.579,-86.956,-50.874,174.723,16.260,152.531
C08004=1090.574,-87.205,-50.863,174.721,16.259,152.531
C08005=1090.568,-87.456,-50.852,174.719,16.258,152.531
C08006=1090.561,-87.705,-50.842,174.717,16.257,152.531
C08007=1090.555,-87.955,-50.831,174.717,16.256,152.531
C08008=1090.549,-88.204,-50.822,174.715,16.256,152.531
C08009=1090.544,-88.454,-50.811,174.713,16.255,152.532
C08010=1090.537,-88.704,-50.801,174.712,16.253,152.532
C08011=1090.531,-88.954,-50.790,174.710,16.253,152.532
C08012=1090.525,-89.203,-50.779,174.708,16.252,152.532
C08013=1090.519,-89.453,-50.769,174.707,16.251,152.532
C08014=1090.513,-89.703,-50.759,174.705,16.251,152.532
C08015=1090.507,-89.953,-50.749,174.704,16.249,152.533
C08016=1090.501,-90.202,-50.738,174.702,16.249,152.533
C08017=1090.495,-90.452,-50.729,174.700,16.248,152.533
C08018=1090.490,-90.701,-50.718,174.699,16.247,152.533
C08019=1090.482,-90.951,-50.707,174.697,16.246,152.533
C08020=1090.477,-91.201,-50.697,174.696,16.245,152.533
C08021=1090.471,-91.450,-50.687,174.694,16.245,152.534
C08022=1090.465,-91.701,-50.676,174.692,16.244,152.534
C08023=1090.459,-91.950,-50.666,174.691,16.242,152.534
C08024=1090.453,-92.200,-50.656,174.690,16.242,152.534
C08025=1090.447,-92.449,-50.645,174.688,16.241,152.534
C08026=1090.441,-92.699,-50.636,174.686,16.241,152.534
C08027=1090.436,-92.949,-50.625,174.684,16.239,152.535
C08028=1090.429,-93.199,-50.615,174.683,16.238,152.535
C08029=1090.423,-93.449,-50.604,174.682,16.238,152.535
C08030=1090.417,-93.698,-50.594,174.680,16.237,152.535
C08031=1090.411,-93.948,-50.583,174.678,16.237,152.535
C08032=1090.405,-94.198,-50.574,174.677,16.235,152.535
C08033=1090.399,-94.447,-50.563,174.675,16.235,152.536
C08034=1090.393,-94.697,-50.553,174.674,16.234,152.536
C08035=1090.388,-94.947,-50.543,174.672,16.233,152.536
C08036=1090.381,-95.196,-50.533,174.670,16.232,152.536
C08037=1090.376,-95.446,-50.523,174.669,16.231,152.536
C08038=1090.369,-95.696,-50.513,174.668,16.231,152.536
C08039=1090.364,-95.946,-50.502,174.666,16.230,152.536
C08040=1090.357,-96.195,-50.492,174.664,16.230,152.537
C08041=1090.351,-96.445,-50.483,174.663,16.228,152.537
C08042=1090.344,-96.721,-50.471,174.661,16.228,152.537
C08043=1090.338,-96.997,-50.460,174.659,16.227,152.537
C08044=1090.332,-97.272,-50.449,174.657,16.226,152.537
C08045=1090.325,-97.548,-50.437,174.655,16.225,152.538
C08046=1090.319,-97.798,-50.428,174.654,16.225,152.538
C08047=1090.313,-98.048,-50.417,174.653,16.224,152.538
C08048=1090.307,-98.297,-50.407,174.651,16.223,152.538
C08049=1090.301,-98.547,-50.398,174.649,16.222,152.538
C08050=1090.295,-98.797,-50.387,174.648,16.222,152.539
C08051=1090.289,-99.047,-50.377,174.646,16.221,152.539
C08052=1090.282,-99.296,-50.368,174.645,16.220,152.539
C08053=1090.277,-99.546,-50.357,174.643,16.219,152.539
C08054=1090.271,-99.796,-50.347,174.642,16.219,152.539
C08055=1090.264,-100.045,-50.338,174.640,16.218,152.539
C08056=1090.258,-100.295,-50.327,174.638,16.217,152.540
C08057=1090.252,-100.545,-50.317,174.636,16.217,152.540
C08058=1090.246,-100.795,-50.307,174.636,16.216,152.540
C08059=1090.239,-101.044,-50.297,174.634,16.215,152.540
C08060=1090.234,-101.295,-50.287,174.632,16.214,152.540
C08061=1090.228,-101.544,-50.277,174.630,16.214,152.541
C08062=1090.221,-101.793,-50.267,174.629,16.213,152.541
C08063=1090.215,-102.043,-50.257,174.627,16.212,152.541
C08064=1090.210,-102.293,-50.247,174.626,16.212,152.541
C08065=1090.203,-102.543,-50.238,174.624,16.211,152.541
C08066=1090.197,-102.792,-50.227,174.623,16.211,152.541
C08067=1090.191,-103.042,-50.218,174.621,16.209,152.542
C08068=1090.185,-103.292,-50.208,174.619,16.209,152.542
C08069=1090.179,-103.542,-50.198,174.617,16.208,152.542
C08070=1090.173,-103.791,-50.188,174.617,16.208,152.542
C08071=1090.166,-104.041,-50.178,174.615,16.207,152.542
C08072=1090.161,-104.291,-50.168,174.613,16.206,152.543
C08073=1090.155,-104.541,-50.158,174.611,16.205,152.543
C08074=1090.148,-104.790,-50.148,174.610,16.205,152.543
C08075=1090.142,-105.040,-50.139,174.608,16.204,152.543
C08076=1090.137,-105.290,-50.128,174.607,16.203,152.543
C08077=1090.131,-105.540,-50.119,174.606,16.203,152.543
C08078=1090.124,-105.790,-50.109,174.604,16.202,152.544
C08079=1090.118,-106.039,-50.099,174.602,16.202,152.544
C08080=1090.112,-106.289,-50.089,174.600,16.200,152.544
C08081=1090.106,-106.539,-50.079,174.599,16.200,152.544
C08082=1090.100,-106.789,-50.070,174.597,16.200,152.545
C08083=1090.094,-107.038,-50.060,174.596,16.199,152.545
C08084=1090.088,-107.288,-50.051,174.595,16.199,152.545
C08085=1090.081,-107.537,-50.040,174.593,16.197,152.545
C08086=1090.075,-107.787,-50.031,174.591,16.197,152.545
C08087=1090.070,-108.037,-50.021,174.589,16.196,152.546
C08088=1090.064,-108.286,-50.011,174.588,16.196,152.546
C08089=1090.058,-108.536,-50.002,174.586,16.195,152.546
C08090=1090.052,-108.786,-49.992,174.585,16.194,152.546
C08091=1090.046,-109.036,-49.983,174.583,16.194,152.546
C08092=1090.039,-109.285,-49.972,174.582,16.193,152.547
C08093=1090.033,-109.535,-49.963,174.580,16.193,152.547
C08094=1090.027,-109.784,-49.953,174.579,16.193,152.547
C08095=1090.021,-110.034,-49.944,174.577,16.191,152.547
C08096=1090.015,-110.284,-49.934,174.575,16.191,152.547
C08097=1090.008,-110.534,-49.925,174.573,16.190,152.548
C08098=1090.002,-110.784,-49.915,174.572,16.190,152.548
C08099=1089.997,-111.034,-49.905,174.571,16.189,152.548
C08100=1089.991,-111.284,-49.895,174.569,16.188,152.548
C08101=1089.984,-111.533,-49.886,174.568,16.188,152.548
C08102=1089.978,-111.783,-49.876,174.566,16.187,152.549
C08103=1089.972,-112.033,-49.867,174.564,16.187,152.549
C08104=1089.966,-112.282,-49.856,174.563,16.187,152.549
C08105=1089.959,-112.532,-49.847,174.561,16.186,152.549
C08106=1089.953,-112.801,-49.837,174.559,16.185,152.549
C08107=1089.947,-113.071,-49.827,174.558,16.184,152.550
C08108=1089.940,-113.340,-49.816,174.556,16.184,152.550
C08109=1089.934,-113.609,-49.806,174.555,16.183,152.550
C08110=1089.927,-113.859,-49.797,174.553,16.183,152.550
C08111=1089.921,-114.109,-49.787,174.551,16.182,152.551
C08112=1089.915,-114.358,-49.778,174.550,16.182,152.551
C08113=1089.909,-114.608,-49.768,174.548,16.181,152.551
C08114=1089.903,-114.858,-49.758,174.546,16.180,152.551
C08115=1089.896,-115.108,-49.749,174.545,16.180,152.551
C08116=1089.890,-115.358,-49.739,174.543,16.179,152.552
C08117=1089.884,-115.607,-49.730,174.541,16.179,152.552
C08118=1089.879,-115.857,-49.721,174.540,16.179,152.552
C08119=1089.872,-116.106,-49.711,174.538,16.178,152.552
C08120=1089.866,-116.356,-49.701,174.537,16.177,152.553
C08121=1089.860,-116.606,-49.692,174.536,16.177,152.553
C08122=1089.854,-116.856,-49.682,174.534,16.176,152.553
C08123=1089.848,-117.106,-49.673,174.532,16.175,152.553
C08124=1089.842,-117.355,-49.663,174.531,16.175,152.553
C08125=1089.835,-117.605,-49.654,174.529,16.175,152.554
C08126=1089.829,-117.855,-49.644,174.527,16.174,152.554
C08127=1089.824,-118.104,-49.635,174.526,16.174,152.554
C08128=1089.817,-118.354,-49.626,174.524,16.173,152.554
C08129=1089.811,-118.604,-49.617,174.523,16.173,152.555
C08130=1089.805,-118.854,-49.607,174.521,16.172,152.555
C08131=1089.799,-119.104,-49.598,174.519,16.172,152.555
C08132=1089.792,-119.353,-49.588,174.518,16.172,152.555
C08133=1089.786,-119.603,-49.579,174.517,16.171,152.555
C08134=1089.780,-119.853,-49.569,174.515,16.170,152.556
C08135=1089.774,-120.102,-49.560,174.514,16.170,152.556
C08136=1089.768,-120.352,-49.550,174.512,16.169,152.556
C08137=1089.762,-120.602,-49.542,174.510,16.169,152.556
C08138=1089.755,-120.852,-49.533,174.509,16.169,152.557
C08139=1089.749,-121.102,-49.523,174.507,16.168,152.557
C08140=1089.743,-121.351,-49.513,174.506,16.168,152.557
C08141=1089.737,-121.601,-49.504,174.504,16.167,152.557
C08142=1089.731,-121.850,-49.495,174.502,16.166,152.558
C08143=1089.726,-122.101,-49.486,174.501,16.166,152.558
C08144=1089.719,-122.350,-49.477,174.499,16.165,152.558
C08145=1089.712,-122.600,-49.467,174.497,16.165,152.558
C08146=1089.706,-122.850,-49.458,174.496,16.165,152.559
C08147=1089.700,-123.100,-49.448,174.494,16.164,152.559
C08148=1089.695,-123.349,-49.440,174.493,16.164,152.559
C08149=1089.689,-123.599,-49.430,174.491,16.163,152.559
C08150=1089.682,-123.849,-49.421,174.489,16.163,152.560
C08151=1089.676,-124.098,-49.412,174.488,16.163,152.560
C08152=1089.669,-124.348,-49.402,174.487,16.162,152.560
C08153=1089.664,-124.598,-49.393,174.485,16.161,152.560
C08154=1089.658,-124.848,-49.384,174.484,16.161,152.560
C08155=1089.651,-125.097,-49.375,174.482,16.160,152.561
C08156=1089.645,-125.347,-49.365,174.480,16.160,152.561
C08157=1089.639,-125.597,-49.357,174.479,16.160,152.561
C08158=1089.633,-125.847,-49.347,174.477,16.159,152.561
C08159=1089.627,-126.096,-49.338,174.476,16.159,152.562
C08160=1089.620,-126.346,-49.329,174.474,16.158,152.562
C08161=1089.615,-126.596,-49.320,174.473,16.158,152.562
C08162=1089.608,-126.846,-49.311,174.471,16.158,152.562
C08163=1089.601,-127.095,-49.301,174.469,16.157,152.563
C08164=1089.596,-127.346,-49.293,174.468,16.157,152.563
C08165=1089.590,-127.595,-49.283,174.466,16.156,152.563
C08166=1089.583,-127.853,-49.274,174.465,16.156,152.563
C08167=1089.577,-128.112,-49.264,174.463,16.156,152.564
C08168=1089.576,-128.370,-49.254,174.461,16.154,152.564
C08169=1089.582,-128.625,-49.240,174.461,16.150,152.563
C08170=1089.177,-128.647,-49.363,174.420,16.256,152.591
C08171=1089.171,-128.391,-49.376,174.420,16.259,152.592
C08172=1089.171,-128.133,-49.387,174.421,16.261,152.592
C08173=1089.177,-127.875,-49.397,174.423,16.262,152.592
C08174=1089.184,-127.617,-49.406,174.424,16.262,152.592
C08175=1089.190,-127.367,-49.415,174.426,16.262,152.591
C08176=1089.196,-127.117,-49.425,174.427,16.262,152.591
C08177=1089.202,-126.868,-49.433,174.429,16.263,152.591
C08178=1089.208,-126.618,-49.442,174.431,16.264,152.591
C08179=1089.215,-126.368,-49.452,174.432,16.264,152.590
C08180=1089.221,-126.118,-49.461,174.434,16.264,152.590
C08181=1089.228,-125.869,-49.470,174.435,16.265,152.590
C08182=1089.233,-125.618,-49.479,174.437,16.266,152.590
C08183=1089.239,-125.369,-49.488,174.439,16.266,152.590
C08184=1089.246,-125.120,-49.497,174.440,16.266,152.589
C08185=1089.252,-124.870,-49.507,174.442,16.267,152.589
C08186=1089.258,-124.620,-49.516,174.443,16.267,152.589
C08187=1089.264,-124.370,-49.525,174.445,16.267,152.589
C08188=1089.270,-124.121,-49.534,174.447,16.268,152.588
C08189=1089.277,-123.871,-49.543,174.448,16.268,152.588
C08190=1089.283,-123.621,-49.552,174.450,16.269,152.588
C08191=1089.289,-123.371,-49.562,174.451,16.269,152.588
C08192=1089.295,-123.121,-49.571,174.452,16.270,152.588
C08193=1089.301,-122.871,-49.581,174.454,16.271,152.587
C08194=1089.307,-122.622,-49.590,174.455,16.271,152.587
C08195=1089.313,-122.372,-49.598,174.457,16.271,152.587
C08196=1089.319,-122.122,-49.608,174.459,16.272,152.586
C08197=1089.326,-121.873,-49.617,174.460,16.272,152.586
C08198=1089.332,-121.623,-49.627,174.462,16.272,152.586
C08199=1089.338,-121.373,-49.637,174.464,16.274,152.586
C08200=1089.343,-121.124,-49.646,174.465,16.274,152.586
C08201=1089.350,-120.874,-49.654,174.467,16.274,152.585
C08202=1089.356,-120.624,-49.664,174.469,16.275,152.585
C08203=1089.362,-120.374,-49.673,174.470,16.275,152.585
C08204=1089.369,-120.124,-49.683,174.472,16.276,152.585
C08205=1089.375,-119.875,-49.692,174.473,16.276,152.585
C08206=1089.381,-119.625,-49.702,174.474,16.277,152.584
C08207=1089.386,-119.376,-49.711,174.476,16.277,152.584
C08208=1089.392,-119.125,-49.720,174.477,16.277,152.584
C08209=1089.399,-118.875,-49.730,174.479,16.278,152.584
C08210=1089.405,-118.626,-49.738,174.481,16.279,152.583
C08211=1089.412,-118.376,-49.748,174.482,16.279,152.583
C08212=1089.418,-118.126,-49.758,174.484,16.280,152.583
C08213=1089.424,-117.877,-49.767,174.486,16.280,152.583
C08214=1089.430,-117.627,-49.777,174.487,16.280,152.582
C08215=1089.436,-117.377,-49.786,174.489,16.281,152.582
C08216=1089.442,-117.128,-49.796,174.491,16.282,152.582
C08217=1089.448,-116.878,-49.805,174.492,16.282,152.582
C08218=1089.454,-116.628,-49.815,174.494,16.283,152.582
C08219=1089.460,-116.378,-49.824,174.495,16.283,152.581
C08220=1089.466,-116.128,-49.833,174.496,16.284,152.581
C08221=1089.472,-115.878,-49.843,174.498,16.285,152.581
C08222=1089.479,-115.628,-49.852,174.500,16.285,152.581
C08223=1089.485,-115.379,-49.862,174.501,16.285,152.581
C08224=1089.491,-115.129,-49.871,174.503,16.286,152.580
C08225=1089.497,-114.879,-49.881,174.505,16.287,152.580
C08226=1089.503,-114.630,-49.890,174.506,16.287,152.580
C08227=1089.509,-114.380,-49.900,174.508,16.288,152.580
C08228=1089.515,-114.130,-49.909,174.509,16.289,152.580
C08229=1089.521,-113.881,-49.919,174.510,16.289,152.579
C08230=1089.527,-113.631,-49.928,174.512,16.290,152.579
C08231=1089.534,-113.361,-49.938,174.514,16.290,152.579
C08232=1089.541,-113.092,-49.949,174.516,16.291,152.579
C08233=1089.547,-112.822,-49.959,174.518,16.292,152.578
C08234=1089.554,-112.552,-49.970,174.519,16.292,152.578
C08235=1089.560,-112.303,-49.979,174.521,16.293,152.578
C08236=1089.566,-112.053,-49.988,174.522,16.294,152.578
C08237=1089.572,-111.804,-49.998,174.524,16.294,152.578
C08238=1089.579,-111.554,-50.007,174.525,16.294,152.577
C08239=1089.584,-111.304,-50.018,174.527,16.295,152.577
C08240=1089.590,-111.054,-50.028,174.529,16.296,152.577
C08241=1089.597,-110.805,-50.037,174.530,16.296,152.577
C08242=1089.603,-110.555,-50.047,174.532,16.297,152.577
C08243=1089.609,-110.305,-50.057,174.534,16.298,152.576
C08244=1089.615,-110.055,-50.066,174.535,16.298,152.576
C08245=1089.621,-109.805,-50.076,174.536,16.299,152.576
C08246=1089.627,-109.556,-50.085,174.538,16.300,152.576
C08247=1089.634,-109.306,-50.095,174.539,16.300,152.576
C08248=1089.640,-109.056,-50.104,174.541,16.301,152.575
C08249=1089.646,-108.806,-50.114,174.543,16.301,152.575
C08250=1089.652,-108.557,-50.124,174.545,16.302,152.575
C08251=1089.658,-108.307,-50.134,174.546,16.303,152.575
C08252=1089.664,-108.057,-50.144,174.548,16.303,152.575
C08253=1089.670,-107.807,-50.154,174.549,16.304,152.574
C08254=1089.676,-107.558,-50.163,174.550,16.304,152.574
C08255=1089.683,-107.308,-50.173,174.552,16.305,152.574
C08256=1089.689,-107.058,-50.182,174.554,16.306,152.574
C08257=1089.695,-106.809,-50.193,174.556,16.307,152.574
C08258=1089.701,-106.559,-50.203,174.557,16.307,152.574
C08259=1089.707,-106.309,-50.212,174.558,16.308,152.573
C08260=1089.713,-106.059,-50.222,174.560,16.309,152.573
C08261=1089.719,-105.809,-50.231,174.561,16.309,152.573
C08262=1089.725,-105.560,-50.241,174.563,16.310,152.573
C08263=1089.731,-105.311,-50.251,174.565,16.311,152.573
C08264=1089.737,-105.061,-50.261,174.567,16.312,152.572
C08265=1089.743,-104.811,-50.271,174.568,16.312,152.572
C08266=1089.749,-104.561,-50.280,174.569,16.313,152.572
C08267=1089.755,-104.312,-50.291,174.571,16.313,152.572
C08268=1089.761,-104.062,-50.301,174.573,16.314,152.572
C08269=1089.767,-103.812,-50.310,174.574,16.314,152.571
C08270=1089.773,-103.562,-50.320,174.576,16.316,152.571
C08271=1089.779,-103.313,-50.329,174.577,16.316,152.571
C08272=1089.785,-103.063,-50.340,174.579,16.317,152.571
C08273=1089.791,-102.813,-50.350,174.580,16.317,152.571
C08274=1089.798,-102.564,-50.359,174.582,16.319,152.571
C08275=1089.803,-102.314,-50.370,174.584,16.319,152.570
C08276=1089.810,-102.064,-50.380,174.585,16.320,152.570
C08277=1089.816,-101.814,-50.390,174.586,16.320,152.570
C08278=1089.822,-101.564,-50.399,174.588,16.321,152.570
C08279=1089.828,-101.314,-50.410,174.590,16.322,152.570
C08280=1089.834,-101.065,-50.420,174.592,16.323,152.569
C08281=1089.840,-100.815,-50.429,174.593,16.323,152.569
C08282=1089.847,-100.566,-50.440,174.595,16.324,152.569
C08283=1089.852,-100.316,-50.450,174.596,16.325,152.569
C08284=1089.859,-100.066,-50.459,174.598,16.326,152.569
C08285=1089.865,-99.817,-50.470,174.599,16.326,152.569
C08286=1089.870,-99.567,-50.480,174.601,16.327,152.568
C08287=1089.877,-99.317,-50.489,174.602,16.328,152.568
C08288=1089.883,-99.068,-50.500,174.604,16.329,152.568
C08289=1089.889,-98.817,-50.510,174.605,16.329,152.568
C08290=1089.895,-98.568,-50.519,174.607,16.330,152.568
C08291=1089.901,-98.318,-50.530,174.609,16.331,152.567
C08292=1089.907,-98.069,-50.539,174.611,16.331,152.567
C08293=1089.913,-97.819,-50.549,174.612,16.333,152.567
C08294=1089.919,-97.569,-50.560,174.613,16.333,152.567
C08295=1089.926,-97.293,-50.571,174.615,16.334,152.567
C08296=1089.932,-97.018,-50.582,174.617,16.335,152.567
C08297=1089.939,-96.741,-50.593,174.619,16.336,152.566
C08298=1089.945,-96.465,-50.604,174.620,16.337,152.566
C08299=1089.952,-96.216,-50.615,174.622,16.337,152.566
C08300=1089.957,-95.966,-50.625,174.624,16.338,152.566
C08301=1089.964,-95.716,-50.635,174.625,16.340,152.566
C08302=1089.970,-95.466,-50.646,174.626,16.340,152.566
C08303=1089.976,-95.216,-50.655,174.628,16.341,152.565
C08304=1089.982,-94.966,-50.666,174.630,16.341,152.565
C08305=1089.988,-94.717,-50.676,174.632,16.342,152.565
C08306=1089.994,-94.467,-50.686,174.633,16.344,152.565
C08307=1090.000,-94.217,-50.696,174.634,16.344,152.565
C08308=1090.005,-93.968,-50.707,174.636,16.345,152.565
C08309=1090.012,-93.718,-50.716,174.638,16.345,152.564
C08310=1090.017,-93.469,-50.727,174.639,16.347,152.564
C08311=1090.024,-93.219,-50.737,174.641,16.348,152.564
C08312=1090.029,-92.969,-50.748,174.642,16.348,152.564
C08313=1090.035,-92.720,-50.757,174.644,16.349,152.564
C08314=1090.041,-92.470,-50.768,174.645,16.350,152.564
C08315=1090.048,-92.220,-50.778,174.647,16.351,152.563
C08316=1090.054,-91.970,-50.789,174.649,16.352,152.563
C08317=1090.060,-91.720,-50.799,174.650,16.352,152.563
C08318=1090.066,-91.471,-50.809,174.652,16.353,152.563
C08319=1090.072,-91.221,-50.819,174.653,16.354,152.563
C08320=1090.078,-90.971,-50.830,174.655,16.355,152.563
C08321=1090.083,-90.721,-50.840,174.657,16.356,152.563
C08322=1090.089,-90.472,-50.850,174.658,16.356,152.562
C08323=1090.095,-90.222,-50.861,174.659,16.357,152.562
C08324=1090.102,-89.972,-50.871,174.661,16.358,152.562
C08325=1090.108,-89.723,-50.882,174.663,16.359,152.562
C08326=1090.114,-89.473,-50.892,174.665,16.360,152.562
C08327=1090.120,-89.223,-50.902,174.666,16.361,152.562
C08328=1090.126,-88.974,-50.912,174.667,16.362,152.562
C08329=1090.132,-88.724,-50.923,174.669,16.363,152.561
C08330=1090.138,-88.475,-50.933,174.671,16.363,152.561
C08331=1090.144,-88.224,-50.944,174.672,16.364,152.561
C08332=1090.150,-87.975,-50.955,174.674,16.366,152.561
C08333=1090.156,-87.725,-50.964,174.675,16.366,152.561
C08334=1090.162,-87.475,-50.975,174.677,16.367,152.561
C08335=1090.168,-87.226,-50.985,174.678,16.368,152.561
C08336=1090.174,-86.976,-50.995,174.680,16.368,152.560
C08337=1090.180,-86.726,-51.007,174.682,16.370,152.560
C08338=1090.186,-86.477,-51.017,174.683,16.371,152.560
C08339=1090.192,-86.227,-51.027,174.685,16.371,152.560
C08340=1090.198,-85.977,-51.037,174.686,16.372,152.560
C08341=1090.204,-85.728,-51.048,174.688,16.373,152.560
C08342=1090.211,-85.477,-51.058,174.690,16.374,152.559
C08343=1090.217,-85.228,-51.069,174.691,16.375,152.559
C08344=1090.222,-84.978,-51.080,174.693,16.376,152.559
C08345=1090.228,-84.729,-51.090,174.694,16.377,152.559
C08346=1090.234,-84.479,-51.100,174.695,16.377,152.559
C08347=1090.241,-84.229,-51.112,174.697,16.378,152.559
C08348=1090.247,-83.980,-51.122,174.699,16.379,152.559
C08349=1090.252,-83.730,-51.132,174.701,16.380,152.558
C08350=1090.259,-83.480,-51.142,174.702,16.381,152.558
C08351=1090.265,-83.230,-51.154,174.704,16.382,152.558
C08352=1090.271,-82.981,-51.165,174.705,16.383,152.558
C08353=1090.277,-82.731,-51.174,174.707,16.383,152.558
C08354=1090.283,-82.482,-51.185,174.708,16.385,152.558
C08355=1090.289,-82.231,-51.196,174.710,16.386,152.558
C08356=1090.296,-81.982,-51.207,174.712,16.386,152.557
C08357=1090.301,-81.732,-51.217,174.713,16.387,152.557
C08358=1090.308,-81.483,-51.227,174.715,16.389,152.557
C08359=1090.314,-81.209,-51.239,174.717,16.390,152.557
C08360=1090.321,-80.935,-51.250,174.718,16.390,152.557
C08361=1090.328,-80.661,-51.263,174.720,16.391,152.557
C08362=1090.335,-80.388,-51.274,174.722,16.393,152.557
C08363=1090.340,-80.138,-51.285,174.724,16.393,152.556
C08364=1090.347,-79.888,-51.295,174.725,16.394,152.556
C08365=1090.352,-79.639,-51.306,174.727,16.395,152.556
C08366=1090.359,-79.389,-51.317,174.728,16.396,152.556
C08367=1090.364,-79.139,-51.328,174.729,16.397,152.556
C08368=1090.370,-78.890,-51.339,174.731,16.398,152.556
C08369=1090.376,-78.640,-51.350,174.733,16.399,152.555
C08370=1090.383,-78.390,-51.359,174.734,16.400,152.555
C08371=1090.388,-78.140,-51.370,174.736,16.401,152.555
C08372=1090.394,-77.891,-51.381,174.738,16.402,152.555
C08373=1090.400,-77.641,-51.392,174.739,16.403,152.555
C08374=1090.406,-77.391,-51.403,174.740,16.404,152.555
C08375=1090.413,-77.142,-51.414,174.742,16.405,152.555
C08376=1090.418,-76.892,-51.425,174.744,16.406,152.555
C08377=1090.424,-76.643,-51.435,174.745,16.407,152.555
C08378=1090.431,-76.393,-51.447,174.747,16.408,152.554
C08379=1090.436,-76.143,-51.457,174.748,16.409,152.554
C08380=1090.442,-75.893,-51.468,174.750,16.410,152.554
C08381=1090.447,-75.644,-51.479,174.752,16.411,152.554
C08382=1090.455,-75.394,-51.489,174.754,16.412,152.554
C08383=1090.460,-75.144,-51.500,174.755,16.413,152.554
C08384=1090.466,-74.895,-51.511,174.756,16.414,152.554
C08385=1090.472,-74.645,-51.522,174.758,16.415,152.554
C08386=1090.478,-74.395,-51.533,174.759,16.416,152.553
C08387=1090.484,-74.146,-51.544,174.761,16.417,152.553
C08388=1090.490,-73.895,-51.555,174.763,16.418,152.553
C08389=1090.496,-73.646,-51.566,174.764,16.419,152.553
C08390=1090.502,-73.396,-51.577,174.766,16.420,152.553
C08391=1090.507,-73.147,-51.588,174.768,16.421,152.553
C08392=1090.513,-72.898,-51.599,174.769,16.422,152.553
C08393=1090.519,-72.647,-51.610,174.771,16.423,152.553
C08394=1090.525,-72.398,-51.621,174.773,16.424,152.552
C08395=1090.531,-72.148,-51.632,174.774,16.426,152.552
C08396=1090.537,-71.898,-51.643,174.775,16.426,152.552
C08397=1090.543,-71.649,-51.654,174.777,16.427,152.552
C08398=1090.549,-71.399,-51.665,174.778,16.428,152.552
C08399=1090.554,-71.150,-51.676,174.780,16.429,152.552
C08400=1090.561,-70.899,-51.687,174.781,16.431,152.552
C08401=1090.567,-70.650,-51.698,174.783,16.432,152.552
C08402=1090.572,-70.401,-51.709,174.785,16.433,152.552
C08403=1090.578,-70.151,-51.719,174.786,16.434,152.552
C08404=1090.584,-69.901,-51.731,174.788,16.435,152.551
C08405=1090.589,-69.651,-51.742,174.790,16.436,152.551
C08406=1090.595,-69.402,-51.753,174.791,16.437,152.551
C08407=1090.601,-69.151,-51.764,174.793,16.438,152.551
C08408=1090.607,-68.902,-51.775,174.795,16.439,152.551
C08409=1090.613,-68.653,-51.787,174.796,16.440,152.551
C08410=1090.620,-68.403,-51.798,174.798,16.441,152.551
C08411=1090.625,-68.153,-51.809,174.800,16.443,152.550
C08412=1090.631,-67.904,-51.820,174.800,16.443,152.550
C08413=1090.637,-67.654,-51.831,174.802,16.444,152.550
C08414=1090.643,-67.404,-51.842,174.804,16.445,152.550
C08415=1090.648,-67.154,-51.853,174.805,16.446,152.550
C08416=1090.654,-66.904,-51.865,174.807,16.448,152.550
C08417=1090.661,-66.655,-51.876,174.808,16.449,152.550
C08418=1090.666,-66.406,-51.887,174.810,16.450,152.550
C08419=1090.673,-66.156,-51.898,174.812,16.451,152.550
C08420=1090.678,-65.906,-51.909,174.813,16.452,152.550
C08421=1090.684,-65.657,-51.920,174.815,16.453,152.549
C08422=1090.690,-65.406,-51.931,174.817,16.454,152.549
C08423=1090.696,-65.135,-51.944,174.818,16.455,152.549
C08424=1090.703,-64.864,-51.956,174.820,16.457,152.549
C08425=1090.710,-64.592,-51.968,174.821,16.458,152.549
C08426=1090.716,-64.321,-51.980,174.823,16.459,152.549
C08427=1090.722,-64.071,-51.992,174.825,16.460,152.549
C08428=1090.727,-63.821,-52.003,174.826,16.461,152.549
C08429=1090.733,-63.572,-52.015,174.828,16.462,152.549
C08430=1090.740,-63.322,-52.026,174.829,16.463,152.549
C08431=1090.746,-63.072,-52.037,174.831,16.465,152.548
C08432=1090.752,-62.822,-52.048,174.833,16.466,152.548
C08433=1090.758,-62.573,-52.060,174.834,16.467,152.548
C08434=1090.763,-62.324,-52.071,174.836,16.468,152.548
C08435=1090.769,-62.073,-52.082,174.838,16.469,152.548
C08436=1090.775,-61.824,-52.093,174.839,16.470,152.548
C08437=1090.782,-61.574,-52.105,174.841,16.471,152.548
C08438=1090.787,-61.325,-52.116,174.842,16.472,152.548
C08439=1090.794,-61.075,-52.127,174.844,16.474,152.548
C08440=1090.799,-60.825,-52.140,174.846,16.475,152.547
C08441=1090.805,-60.575,-52.151,174.847,16.476,152.547
C08442=1090.811,-60.326,-52.162,174.849,16.477,152.547
C08443=1090.817,-60.076,-52.173,174.850,16.478,152.547
C08444=1090.824,-59.827,-52.185,174.852,16.479,152.547
C08445=1090.829,-59.577,-52.196,174.854,16.480,152.547
C08446=1090.835,-59.327,-52.208,174.855,16.481,152.547
C08447=1090.841,-59.078,-52.219,174.857,16.483,152.547
C08448=1090.847,-58.828,-52.230,174.859,16.484,152.547
C08449=1090.853,-58.579,-52.242,174.860,16.485,152.546
C08450=1090.859,-58.328,-52.254,174.862,16.486,152.546
C08451=1090.865,-58.079,-52.264,174.863,16.487,152.546
C08452=1090.871,-57.829,-52.276,174.865,16.488,152.546
C08453=1090.877,-57.580,-52.287,174.867,16.489,152.546
C08454=1090.883,-57.330,-52.300,174.868,16.490,152.546
C08455=1090.889,-57.080,-52.311,174.870,16.492,152.546
C08456=1090.895,-56.830,-52.322,174.872,16.493,152.546
C08457=1090.901,-56.581,-52.334,174.873,16.494,152.546
C08458=1090.907,-56.331,-52.345,174.875,16.495,152.546
C08459=1090.913,-56.082,-52.357,174.876,16.496,152.545
C08460=1090.919,-55.832,-52.368,174.878,16.497,152.545
C08461=1090.925,-55.583,-52.380,174.880,16.498,152.545
C08462=1090.931,-55.333,-52.391,174.881,16.499,152.545
C08463=1090.937,-55.083,-52.403,174.883,16.501,152.545
C08464=1090.943,-54.833,-52.414,174.884,16.502,152.545
C08465=1090.949,-54.583,-52.426,174.886,16.503,152.545
C08466=1090.955,-54.334,-52.437,174.888,16.504,152.545
C08467=1090.961,-54.084,-52.449,174.889,16.505,152.545
C08468=1090.967,-53.835,-52.461,174.891,16.506,152.544
C08469=1090.973,-53.585,-52.472,174.893,16.507,152.544
C08470=1090.979,-53.335,-52.484,174.894,16.509,152.544
C08471=1090.985,-53.085,-52.495,174.896,16.510,152.544
C08472=1090.991,-52.836,-52.507,174.897,16.511,152.544
C08473=1090.998,-52.587,-52.519,174.899,16.512,152.544
C08474=1091.003,-52.336,-52.531,174.901,16.513,152.544
C08475=1091.009,-52.087,-52.542,174.902,16.514,152.544
C08476=1091.016,-51.837,-52.554,174.904,16.515,152.544
C08477=1091.021,-51.588,-52.566,174.905,16.516,152.544
C08478=1091.027,-51.338,-52.577,174.907,16.518,152.543
C08479=1091.034,-51.088,-52.589,174.909,16.519,152.543
C08480=1091.040,-50.839,-52.601,174.910,16.520,152.543
C08481=1091.046,-50.589,-52.612,174.912,16.521,152.543
C08482=1091.052,-50.340,-52.624,174.913,16.523,152.543
C08483=1091.057,-50.090,-52.636,174.915,16.524,152.543
C08484=1091.063,-49.841,-52.648,174.917,16.525,152.543
C08485=1091.069,-49.590,-52.659,174.918,16.526,152.543
C08486=1091.076,-49.341,-52.671,174.920,16.527,152.543
C08487=1091.081,-49.071,-52.685,174.922,16.529,152.543
C08488=1091.088,-48.800,-52.697,174.924,16.530,152.542
C08489=1091.094,-48.530,-52.710,174.925,16.532,152.543
C08490=1091.101,-48.260,-52.722,174.927,16.533,152.542
C08491=1091.106,-48.011,-52.734,174.928,16.534,152.542
C08492=1091.113,-47.761,-52.746,174.930,16.535,152.542
C08493=1091.118,-47.511,-52.758,174.932,16.536,152.542
C08494=1091.124,-47.261,-52.770,174.933,16.537,152.542
C08495=1091.130,-47.012,-52.782,174.935,16.538,152.542
C08496=1091.135,-46.762,-52.794,174.937,16.541,152.542
C08497=1091.142,-46.512,-52.806,174.939,16.542,152.542
C08498=1091.147,-46.263,-52.818,174.940,16.543,152.542
C08499=1091.154,-46.013,-52.829,174.942,16.544,152.542
C08500=1091.160,-45.763,-52.842,174.943,16.545,152.542
C08501=1091.166,-45.514,-52.853,174.945,16.546,152.541
C08502=1091.171,-45.264,-52.866,174.947,16.547,152.541
C08503=1091.176,-45.015,-52.877,174.948,16.549,152.541
C08504=1091.183,-44.765,-52.889,174.950,16.550,152.541
C08505=1091.189,-44.515,-52.902,174.951,16.551,152.541
C08506=1091.195,-44.266,-52.913,174.953,16.552,152.541
C08507=1091.201,-44.016,-52.925,174.955,16.553,152.541
C08508=1091.206,-43.767,-52.938,174.956,16.555,152.541
C08509=1091.213,-43.517,-52.950,174.958,16.556,152.541
C08510=1091.219,-43.267,-52.962,174.959,16.557,152.541
C08511=1091.224,-43.018,-52.973,174.961,16.558,152.541
C08512=1091.230,-42.768,-52.986,174.963,16.560,152.541
C08513=1091.236,-42.518,-52.998,174.965,16.561,152.540
C08514=1091.242,-42.269,-53.010,174.966,16.562,152.540
C08515=1091.248,-42.019,-53.022,174.968,16.564,152.540
C08516=1091.254,-41.769,-53.034,174.970,16.565,152.540
C08517=1091.260,-41.520,-53.046,174.971,16.566,152.540
C08518=1091.266,-41.270,-53.058,174.973,16.567,152.540
C08519=1091.272,-41.020,-53.070,174.974,16.569,152.540
C08520=1091.278,-40.771,-53.082,174.976,16.570,152.540
C08521=1091.283,-40.521,-53.095,174.977,16.571,152.540
C08522=1091.290,-40.271,-53.106,174.979,16.572,152.540
C08523=1091.295,-40.022,-53.118,174.981,16.573,152.540
C08524=1091.301,-39.772,-53.131,174.982,16.574,152.539
C08525=1091.308,-39.522,-53.143,174.984,16.576,152.539
C08526=1091.313,-39.273,-53.155,174.986,16.577,152.539
C08527=1091.319,-39.023,-53.168,174.988,16.579,152.539
C08528=1091.326,-38.774,-53.180,174.989,16.580,152.539
C08529=1091.331,-38.525,-53.192,174.991,16.581,152.539
C08530=1091.337,-38.275,-53.204,174.992,16.582,152.539
C08531=1091.342,-38.024,-53.216,174.994,16.584,152.539
C08532=1091.348,-37.775,-53.228,174.995,16.585,152.539
C08533=1091.354,-37.525,-53.240,174.997,16.586,152.539
C08534=1091.360,-37.276,-53.253,174.999,16.587,152.539
C08535=1091.366,-37.026,-53.265,175.000,16.589,152.539
C08536=1091.371,-36.777,-53.278,175.002,16.590,152.539
C08537=1091.378,-36.527,-53.290,175.004,16.591,152.538
C08538=1091.383,-36.278,-53.302,175.006,16.593,152.538
C08539=1091.389,-36.028,-53.314,175.007,16.594,152.538
C08540=1091.395,-35.778,-53.327,175.009,16.595,152.538
C08541=1091.401,-35.528,-53.339,175.010,16.596,152.538
C08542=1091.406,-35.279,-53.352,175.012,16.598,152.538
C08543=1091.413,-35.029,-53.364,175.013,16.599,152.538
C08544=1091.419,-34.779,-53.376,175.015,16.600,152.538
C08545=1091.424,-34.530,-53.388,175.016,16.602,152.538
C08546=1091.430,-34.280,-53.401,175.019,16.603,152.538
C08547=1091.436,-34.031,-53.413,175.020,16.604,152.538
C08548=1091.442,-33.781,-53.426,175.022,16.605,152.538
C08549=1091.447,-33.531,-53.438,175.024,16.607,152.537
C08550=1091.454,-33.282,-53.450,175.025,16.608,152.538
C08551=1091.460,-33.012,-53.464,175.027,16.609,152.537
C08552=1091.467,-32.742,-53.477,175.029,16.611,152.537
C08553=1091.472,-32.473,-53.491,175.031,16.612,152.537
C08554=1091.479,-32.203,-53.504,175.032,16.613,152.537
C08555=1091.485,-31.953,-53.516,175.034,16.615,152.537
C08556=1091.491,-31.703,-53.529,175.035,16.616,152.537
C08557=1091.497,-31.454,-53.542,175.038,16.618,152.537
C08558=1091.503,-31.204,-53.554,175.039,16.619,152.537
C08559=1091.508,-30.955,-53.567,175.041,16.620,152.537
C08560=1091.514,-30.705,-53.579,175.042,16.622,152.537
C08561=1091.520,-30.455,-53.592,175.044,16.623,152.537
C08562=1091.526,-30.206,-53.604,175.046,16.624,152.537
C08563=1091.532,-29.956,-53.617,175.047,16.625,152.536
C08564=1091.538,-29.706,-53.629,175.049,16.626,152.536
C08565=1091.544,-29.457,-53.642,175.051,16.628,152.536
C08566=1091.550,-29.207,-53.655,175.052,16.629,152.536
C08567=1091.556,-28.958,-53.667,175.054,16.631,152.536
C08568=1091.562,-28.708,-53.679,175.056,16.632,152.536
C08569=1091.567,-28.458,-53.692,175.057,16.633,152.536
C08570=1091.574,-28.209,-53.705,175.059,16.634,152.536
C08571=1091.580,-27.959,-53.718,175.060,16.636,152.536
C08572=1091.585,-27.709,-53.730,175.062,16.637,152.536
C08573=1091.591,-27.460,-53.742,175.064,16.638,152.536
C08574=1091.597,-27.210,-53.755,175.066,16.640,152.536
C08575=1091.603,-26.961,-53.768,175.068,16.641,152.535
C08576=1091.609,-26.711,-53.781,175.069,16.642,152.535
C08577=1091.615,-26.461,-53.793,175.071,16.643,152.535
C08578=1091.620,-26.212,-53.805,175.072,16.645,152.535
C08579=1091.626,-25.962,-53.819,175.074,16.646,152.535
C08580=1091.632,-25.713,-53.831,175.076,16.648,152.535
C08581=1091.638,-25.463,-53.844,175.078,16.649,152.535
C08582=1091.644,-25.213,-53.856,175.079,16.650,152.535
C08583=1091.650,-24.964,-53.869,175.081,16.651,152.535
C08584=1091.655,-24.714,-53.882,175.082,16.653,152.535
C08585=1091.661,-24.464,-53.895,175.084,16.654,152.535
C08586=1091.667,-24.215,-53.908,175.085,16.655,152.535
C08587=1091.673,-23.965,-53.921,175.088,16.657,152.535
C08588=1091.679,-23.715,-53.933,175.089,16.658,152.535
C08589=1091.684,-23.467,-53.946,175.091,16.660,152.535
C08590=1091.690,-23.217,-53.959,175.092,16.661,152.534
C08591=1091.696,-22.967,-53.971,175.094,16.662,152.534
C08592=1091.702,-22.717,-53.985,175.095,16.664,152.534
C08593=1091.707,-22.467,-53.998,175.098,16.665,152.534
C08594=1091.713,-22.217,-54.010,175.099,16.666,152.534
C08595=1091.720,-21.968,-54.024,175.101,16.667,152.534
C08596=1091.725,-21.719,-54.036,175.102,16.669,152.534
C08597=1091.731,-21.469,-54.048,175.104,16.670,152.534
C08598=1091.737,-21.220,-54.062,175.106,16.671,152.534
C08599=1091.742,-20.970,-54.075,175.108,16.673,152.534
C08600=1091.748,-20.720,-54.088,175.109,16.675,152.534
C08601=1091.754,-20.471,-54.101,175.111,16.676,152.534
C08602=1091.760,-20.221,-54.113,175.113,16.677,152.534
C08603=1091.766,-19.971,-54.126,175.114,16.678,152.533
C08604=1091.772,-19.722,-54.139,175.116,16.679,152.533
C08605=1091.777,-19.473,-54.153,175.118,16.681,152.533
C08606=1091.783,-19.223,-54.165,175.120,16.682,152.533
C08607=1091.789,-18.974,-54.178,175.121,16.684,152.533
C08608=1091.795,-18.724,-54.191,175.123,16.685,152.533
C08609=1091.801,-18.474,-54.204,175.124,16.686,152.533
C08610=1091.807,-18.224,-54.217,175.126,16.688,152.533
C08611=1091.813,-17.975,-54.231,175.128,16.689,152.533
C08612=1091.819,-17.725,-54.243,175.130,16.690,152.533
C08613=1091.825,-17.476,-54.256,175.131,16.691,152.533
C08614=1091.831,-17.226,-54.269,175.133,16.693,152.533
C08615=1091.836,-16.955,-54.283,175.135,16.695,152.533
C08616=1091.843,-16.685,-54.298,175.137,16.696,152.532
C08617=1091.850,-16.414,-54.312,175.138,16.697,152.532
C08618=1091.856,-16.144,-54.326,175.141,16.699,152.532
C08619=1091.862,-15.894,-54.339,175.142,16.700,152.532
C08620=1091.867,-15.644,-54.352,175.144,16.701,152.532
C08621=1091.873,-15.395,-54.365,175.145,16.703,152.532
C08622=1091.879,-15.145,-54.378,175.147,16.704,152.532
C08623=1091.885,-14.896,-54.391,175.149,16.706,152.532
C08624=1091.891,-14.645,-54.404,175.151,16.707,152.532
C08625=1091.897,-14.396,-54.417,175.152,16.708,152.532
C08626=1091.902,-14.147,-54.431,175.154,16.709,152.532
C08627=1091.908,-13.897,-54.444,175.155,16.711,152.532
C08628=1091.914,-13.647,-54.457,175.158,16.713,152.532
C08629=1091.920,-13.397,-54.470,175.159,16.714,152.532
C08630=1091.926,-13.148,-54.484,175.161,16.715,152.531
C08631=1091.932,-12.899,-54.497,175.162,16.717,152.531
C08632=1091.937,-12.649,-54.510,175.164,16.718,152.531
C08633=1091.943,-12.399,-54.523,175.166,16.719,152.531
C08634=1091.949,-12.150,-54.537,175.168,16.720,152.531
C08635=1091.955,-11.900,-54.550,175.169,16.722,152.531
C08636=1091.960,-11.650,-54.564,175.171,16.723,152.531
C08637=1091.967,-11.401,-54.577,175.173,16.724,152.531
C08638=1091.972,-11.151,-54.589,175.175,16.726,152.531
C08639=1091.978,-10.902,-54.603,175.176,16.728,152.531
C08640=1091.984,-10.652,-54.617,175.178,16.729,152.531
C08641=1091.989,-10.402,-54.630,175.180,16.730,152.531
C08642=1091.996,-10.153,-54.643,175.181,16.731,152.531
C08643=1092.001,-9.903,-54.657,175.183,16.733,152.531
C08644=1092.007,-9.654,-54.670,175.185,16.734,152.530
C08645=1092.013,-9.404,-54.683,175.187,16.735,152.530
C08646=1092.019,-9.155,-54.696,175.188,16.737,152.530
C08647=1092.025,-8.905,-54.710,175.190,16.738,152.530
C08648=1092.030,-8.656,-54.724,175.192,16.740,152.530
C08649=1092.036,-8.406,-54.736,175.194,16.741,152.530
C08650=1092.042,-8.156,-54.750,175.195,16.742,152.530
C08651=1092.048,-7.907,-54.763,175.197,16.743,152.530
C08652=1092.053,-7.657,-54.777,175.199,16.746,152.530
C08653=1092.060,-7.408,-54.790,175.201,16.747,152.530
C08654=1092.065,-7.158,-54.804,175.202,16.748,152.530
C08655=1092.071,-6.909,-54.817,175.204,16.749,152.530
C08656=1092.076,-6.659,-54.831,175.205,16.750,152.530
C08657=1092.083,-6.410,-54.844,175.208,16.752,152.530
C08658=1092.088,-6.160,-54.858,175.209,16.753,152.529
C08659=1092.094,-5.910,-54.870,175.211,16.754,152.529
C08660=1092.099,-5.661,-54.884,175.212,16.756,152.529
C08661=1092.106,-5.411,-54.898,175.215,16.757,152.529
C08662=1092.112,-5.161,-54.912,175.216,16.759,152.529
C08663=1092.118,-4.912,-54.925,175.218,16.760,152.529
C08664=1092.123,-4.662,-54.939,175.219,16.761,152.529
C08665=1092.130,-4.413,-54.952,175.221,16.762,152.529
C08666=1092.135,-4.164,-54.966,175.224,16.764,152.529
C08667=1092.141,-3.914,-54.979,175.225,16.765,152.529
C08668=1092.147,-3.664,-54.992,175.226,16.767,152.529
C08669=1092.153,-3.415,-55.006,175.228,16.768,152.529
C08670=1092.159,-3.165,-55.020,175.231,16.770,152.528
C08671=1092.164,-2.915,-55.034,175.232,16.771,152.528
C08672=1092.171,-2.666,-55.047,175.233,16.772,152.528
C08673=1092.176,-2.416,-55.061,175.235,16.773,152.528
C08674=1092.181,-2.167,-55.075,175.238,16.775,152.528
C08675=1092.188,-1.917,-55.088,175.239,16.776,152.528
C08676=1092.193,-1.668,-55.102,175.240,16.778,152.528
C08677=1092.199,-1.418,-55.116,175.242,16.779,152.528
C08678=1092.204,-1.169,-55.130,175.245,16.781,152.528
C08679=1092.211,-0.897,-55.145,175.246,16.782,152.528
C08680=1092.217,-0.624,-55.159,175.248,16.783,152.528
C08681=1092.223,-0.352,-55.174,175.250,16.785,152.528
C08682=1092.229,-0.080,-55.189,175.252,16.786,152.528
C08683=1092.235,0.170,-55.203,175.254,16.788,152.527
C08684=1092.241,0.419,-55.217,175.255,16.790,152.527
C08685=1092.247,0.670,-55.231,175.257,16.791,152.527
C08686=1092.252,0.919,-55.245,175.259,16.792,152.527
C08687=1092.258,1.169,-55.259,175.261,16.794,152.527
C08688=1092.264,1.418,-55.272,175.262,16.795,152.527
C08689=1092.269,1.668,-55.286,175.264,16.796,152.527
C08690=1092.275,1.917,-55.300,175.266,16.797,152.527
C08691=1092.280,2.167,-55.313,175.268,16.799,152.527
C08692=1092.287,2.416,-55.327,175.269,16.801,152.527
C08693=1092.293,2.666,-55.341,175.271,16.802,152.527
C08694=1092.298,2.915,-55.355,175.273,16.803,152.527
C08695=1092.304,3.165,-55.369,175.275,16.805,152.527
C08696=1092.309,3.414,-55.383,175.277,16.806,152.526
C08697=1092.316,3.664,-55.396,175.278,16.807,152.527
C08698=1092.321,3.913,-55.410,175.280,16.809,152.526
C08699=1092.327,4.164,-55.425,175.282,16.810,152.526
C08700=1092.333,4.413,-55.438,175.284,16.811,152.526
C08701=1092.338,4.663,-55.452,175.285,16.813,152.526
C08702=1092.345,4.911,-55.466,175.287,16.815,152.526
C08703=1092.350,5.161,-55.480,175.289,16.816,152.526
C08704=1092.356,5.410,-55.494,175.291,16.817,152.526
C08705=1092.362,5.661,-55.508,175.292,16.818,152.526
C08706=1092.367,5.910,-55.522,175.295,16.820,152.526
C08707=1092.373,6.159,-55.537,175.296,16.821,152.526
C08708=1092.379,6.409,-55.550,175.298,16.823,152.526
C08709=1092.385,6.659,-55.564,175.299,16.824,152.526
C08710=1092.391,6.908,-55.578,175.302,16.825,152.525
C08711=1092.396,7.158,-55.592,175.303,16.826,152.525
C08712=1092.402,7.407,-55.606,175.305,16.828,152.525
C08713=1092.407,7.656,-55.620,175.307,16.829,152.525
C08714=1092.414,7.907,-55.635,175.309,16.831,152.525
C08715=1092.420,8.156,-55.648,175.310,16.832,152.525
C08716=1092.426,8.405,-55.662,175.312,16.833,152.525
C08717=1092.431,8.655,-55.676,175.314,16.835,152.525
C08718=1092.437,8.905,-55.691,175.316,16.836,152.525
C08719=1092.443,9.154,-55.705,175.318,16.837,152.525
C08720=1092.448,9.403,-55.719,175.319,16.838,152.524
C08721=1092.454,9.654,-55.733,175.321,16.840,152.524
C08722=1092.460,9.903,-55.748,175.323,16.842,152.524
C08723=1092.466,10.152,-55.761,175.325,16.843,152.524
C08724=1092.472,10.401,-55.775,175.327,16.844,152.524
C08725=1092.478,10.651,-55.790,175.329,16.846,152.524
C08726=1092.484,10.901,-55.804,175.330,16.847,152.524
C08727=1092.489,11.150,-55.818,175.332,16.848,152.524
C08728=1092.496,11.400,-55.833,175.334,16.849,152.524
C08729=1092.501,11.649,-55.846,175.336,16.851,152.524
C08730=1092.507,11.899,-55.860,175.337,16.852,152.524
C08731=1092.512,12.148,-55.875,175.340,16.854,152.524
C08732=1092.518,12.398,-55.889,175.341,16.855,152.523
C08733=1092.524,12.647,-55.904,175.343,16.856,152.523
C08734=1092.530,12.896,-55.917,175.345,16.857,152.523
C08735=1092.536,13.147,-55.931,175.347,16.859,152.523
C08736=1092.542,13.396,-55.946,175.349,16.860,152.523
C08737=1092.548,13.646,-55.960,175.350,16.861,152.523
C08738=1092.554,13.895,-55.975,175.353,16.863,152.523
C08739=1092.560,14.145,-55.988,175.354,16.864,152.523
C08740=1092.566,14.394,-56.003,175.356,16.865,152.523
C08741=1092.571,14.644,-56.017,175.357,16.867,152.523
C08742=1092.577,14.893,-56.032,175.360,16.869,152.522
C08743=1092.583,15.167,-56.048,175.361,16.870,152.522
C08744=1092.590,15.442,-56.064,175.364,16.871,152.522
C08745=1092.596,15.716,-56.079,175.365,16.872,152.522
C08746=1092.602,15.990,-56.095,175.368,16.874,152.522
C08747=1092.608,16.240,-56.110,175.369,16.875,152.522
C08748=1092.614,16.490,-56.124,175.372,16.877,152.522
C08749=1092.619,16.738,-56.138,175.373,16.879,152.522
C08750=1092.625,16.989,-56.153,175.375,16.880,152.522
C08751=1092.631,17.238,-56.167,175.376,16.881,152.522
C08752=1092.637,17.487,-56.181,175.379,16.883,152.521
C08753=1092.642,17.737,-56.197,175.381,16.884,152.521
C08754=1092.648,17.987,-56.210,175.382,16.885,152.521
C08755=1092.654,18.236,-56.225,175.385,16.886,152.521
C08756=1092.660,18.485,-56.240,175.386,16.888,152.521
C08757=1092.665,18.735,-56.254,175.388,16.889,152.521
C08758=1092.672,18.985,-56.269,175.390,16.890,152.521
C08759=1092.677,19.234,-56.283,175.392,16.892,152.521
C08760=1092.682,19.484,-56.298,175.393,16.893,152.521
C08761=1092.689,19.733,-56.313,175.396,16.895,152.521
C08762=1092.694,19.983,-56.327,175.397,16.896,152.521
C08763=1092.701,20.232,-56.342,175.399,16.897,152.520
C08764=1092.706,20.481,-56.356,175.401,16.899,152.520
C08765=1092.712,20.731,-56.370,175.403,16.900,152.520
C08766=1092.718,20.981,-56.385,175.405,16.901,152.520
C08767=1092.723,21.230,-56.399,175.407,16.903,152.520
C08768=1092.729,21.479,-56.414,175.409,16.904,152.520
C08769=1092.734,21.729,-56.429,175.410,16.905,152.520
C08770=1092.740,21.978,-56.444,175.412,16.906,152.520
C08771=1092.746,22.229,-56.458,175.414,16.908,152.520
C08772=1092.752,22.478,-56.473,175.416,16.909,152.520
C08773=1092.757,22.727,-56.488,175.417,16.911,152.520
C08774=1092.763,22.977,-56.502,175.420,16.912,152.519
C08775=1092.769,23.226,-56.517,175.421,16.913,152.519
C08776=1092.775,23.476,-56.532,175.423,16.915,152.519
C08777=1092.780,23.725,-56.547,175.425,16.916,152.519
C08778=1092.786,23.975,-56.561,175.427,16.917,152.519
C08779=1092.792,24.224,-56.576,175.429,16.918,152.519
C08780=1092.797,24.473,-56.591,175.431,16.920,152.519
C08781=1092.804,24.723,-56.606,175.433,16.921,152.519
C08782=1092.809,24.973,-56.620,175.434,16.922,152.519
C08783=1092.816,25.222,-56.635,175.437,16.924,152.518
C08784=1092.821,25.472,-56.650,175.438,16.925,152.518
C08785=1092.827,25.721,-56.665,175.441,16.927,152.518
C08786=1092.833,25.970,-56.679,175.442,16.928,152.518
C08787=1092.838,26.220,-56.695,175.444,16.929,152.518
C08788=1092.844,26.470,-56.709,175.446,16.931,152.518
C08789=1092.850,26.719,-56.724,175.448,16.932,152.518
C08790=1092.855,26.969,-56.739,175.450,16.933,152.518
C08791=1092.862,27.218,-56.754,175.452,16.935,152.518
C08792=1092.867,27.467,-56.768,175.454,16.936,152.517
C08793=1092.873,27.717,-56.784,175.455,16.937,152.517
C08794=1092.879,27.966,-56.799,175.458,16.939,152.517
C08795=1092.884,28.217,-56.813,175.459,16.940,152.517
C08796=1092.890,28.466,-56.828,175.461,16.941,152.517
C08797=1092.896,28.715,-56.843,175.463,16.943,152.517
C08798=1092.901,28.965,-56.858,175.465,16.944,152.517
C08799=1092.908,29.214,-56.873,175.467,16.945,152.517
C08800=1092.913,29.464,-56.888,175.469,16.947,152.517
C08801=1092.919,29.713,-56.903,175.471,16.948,152.516
C08802=1092.924,29.963,-56.918,175.472,16.949,152.516
C08803=1092.930,30.212,-56.933,175.475,16.951,152.516
C08804=1092.936,30.462,-56.948,175.476,16.952,152.516
C08805=1092.941,30.710,-56.963,175.479,16.953,152.516
C08806=1092.947,30.960,-56.979,175.481,16.955,152.516
C08807=1092.954,31.236,-56.995,175.482,16.956,152.516
C08808=1092.960,31.512,-57.011,175.485,16.957,152.516
C08809=1092.966,31.788,-57.028,175.487,16.959,152.515
C08810=1092.973,32.064,-57.045,175.489,16.960,152.515
C08811=1092.978,32.313,-57.060,175.491,16.962,152.515
C08812=1092.984,32.563,-57.075,175.493,16.963,152.515
C08813=1092.989,32.812,-57.090,175.494,16.964,152.515
C08814=1092.996,33.062,-57.105,175.497,16.966,152.515
C08815=1093.001,33.311,-57.120,175.498,16.967,152.515
C08816=1093.007,33.561,-57.135,175.501,16.969,152.515
C08817=1093.012,33.810,-57.151,175.502,16.970,152.515
C08818=1093.018,34.060,-57.165,175.504,16.971,152.515
C08819=1093.024,34.308,-57.181,175.507,16.972,152.514
C08820=1093.030,34.558,-57.196,175.508,16.973,152.514
C08821=1093.036,34.808,-57.212,175.510,16.974,152.514
C08822=1093.042,35.057,-57.226,175.512,16.976,152.514
C08823=1093.047,35.307,-57.242,175.514,16.977,152.514
C08824=1093.052,35.556,-57.257,175.516,16.978,152.514
C08825=1093.059,35.806,-57.272,175.518,16.980,152.514
C08826=1093.064,36.056,-57.288,175.520,16.981,152.513
C08827=1093.070,36.304,-57.303,175.522,16.983,152.513
C08828=1093.076,36.554,-57.318,175.524,16.984,152.513
C08829=1093.082,36.803,-57.333,175.526,16.985,152.513
C08830=1093.087,37.053,-57.349,175.528,16.986,152.513
C08831=1093.093,37.303,-57.364,175.530,16.987,152.513
C08832=1093.099,37.552,-57.379,175.532,16.989,152.513
C08833=1093.105,37.801,-57.395,175.534,16.990,152.513
C08834=1093.110,38.051,-57.411,175.535,16.991,152.512
C08835=1093.116,38.300,-57.425,175.538,16.993,152.512
C08836=1093.122,38.550,-57.441,175.539,16.994,152.512
C08837=1093.127,38.799,-57.456,175.541,16.995,152.512
C08838=1093.134,39.048,-57.471,175.544,16.997,152.512
C08839=1093.139,39.298,-57.487,175.545,16.998,152.512
C08840=1093.144,39.548,-57.502,175.548,16.999,152.512
C08841=1093.150,39.798,-57.518,175.549,17.000,152.512
C08842=1093.156,40.046,-57.533,175.551,17.002,152.511
C08843=1093.162,40.296,-57.549,175.554,17.003,152.511
C08844=1093.167,40.546,-57.564,175.555,17.004,152.511
C08845=1093.173,40.794,-57.580,175.558,17.006,152.511
C08846=1093.179,41.044,-57.595,175.559,17.007,152.511
C08847=1093.185,41.294,-57.610,175.561,17.008,152.511
C08848=1093.190,41.543,-57.626,175.564,17.010,152.511
C08849=1093.196,41.793,-57.642,175.565,17.011,152.510
C08850=1093.201,42.042,-57.657,175.568,17.012,152.510
C08851=1093.207,42.291,-57.673,175.569,17.014,152.510
C08852=1093.213,42.541,-57.688,175.571,17.015,152.510
C08853=1093.218,42.790,-57.703,175.574,17.016,152.510
C08854=1093.224,43.040,-57.720,175.575,17.017,152.510
C08855=1093.230,43.289,-57.735,175.578,17.019,152.510
C08856=1093.236,43.539,-57.750,175.579,17.020,152.510
C08857=1093.241,43.788,-57.766,175.581,17.021,152.509
C08858=1093.247,44.038,-57.782,175.583,17.023,152.509
C08859=1093.252,44.286,-57.798,175.585,17.023,152.509
C08860=1093.258,44.536,-57.813,175.588,17.025,152.509
C08861=1093.264,44.786,-57.829,175.589,17.026,152.509
C08862=1093.269,45.035,-57.844,175.591,17.027,152.509
C08863=1093.275,45.285,-57.860,175.593,17.029,152.509
C08864=1093.281,45.534,-57.876,175.595,17.030,152.509
C08865=1093.286,45.784,-57.891,175.597,17.032,152.508
C08866=1093.292,46.033,-57.908,175.599,17.032,152.508
C08867=1093.297,46.283,-57.923,175.602,17.034,152.508
C08868=1093.303,46.532,-57.939,175.603,17.035,152.508
C08869=1093.308,46.782,-57.955,175.605,17.036,152.508
C08870=1093.314,47.032,-57.970,175.607,17.038,152.508
C08871=1093.321,47.306,-57.987,175.610,17.040,152.508
C08872=1093.327,47.583,-58.005,175.612,17.040,152.507
C08873=1093.333,47.858,-58.023,175.614,17.042,152.507
C08874=1093.339,48.134,-58.040,175.617,17.044,152.507
C08875=1093.345,48.383,-58.056,175.618,17.045,152.507
C08876=1093.351,48.633,-58.072,175.620,17.046,152.507
C08877=1093.356,48.882,-58.088,175.623,17.047,152.507
C08878=1093.362,49.132,-58.103,175.624,17.048,152.506
C08879=1093.367,49.381,-58.119,175.627,17.050,152.506
C08880=1093.373,49.631,-58.135,175.628,17.051,152.506
C08881=1093.378,49.880,-58.151,175.631,17.052,152.506
C08882=1093.384,50.129,-58.167,175.633,17.053,152.506
C08883=1093.390,50.379,-58.183,175.634,17.055,152.506
C08884=1093.396,50.628,-58.199,175.637,17.056,152.506
C08885=1093.401,50.877,-58.214,175.639,17.057,152.505
C08886=1093.407,51.127,-58.230,175.641,17.059,152.505
C08887=1093.413,51.376,-58.247,175.643,17.060,152.505
C08888=1093.419,51.626,-58.262,175.645,17.061,152.505
C08889=1093.425,51.876,-58.278,175.647,17.062,152.505
C08890=1093.430,52.124,-58.294,175.649,17.063,152.505
C08891=1093.435,52.374,-58.310,175.651,17.065,152.505
C08892=1093.441,52.624,-58.327,175.653,17.066,152.504
C08893=1093.447,52.873,-58.343,175.655,17.067,152.504
C08894=1093.452,53.123,-58.359,175.657,17.068,152.504
C08895=1093.458,53.372,-58.374,175.660,17.070,152.504
C08896=1093.464,53.621,-58.391,175.661,17.071,152.504
C08897=1093.470,53.870,-58.407,175.664,17.072,152.504
C08898=1093.475,54.120,-58.422,175.666,17.073,152.503
C08899=1093.481,54.370,-58.439,175.667,17.074,152.503
C08900=1093.487,54.619,-58.455,175.670,17.076,152.503
C08901=1093.493,54.868,-58.471,175.672,17.076,152.503
C08902=1093.497,55.118,-58.487,175.674,17.078,152.503
C08903=1093.503,55.367,-58.503,175.676,17.079,152.503
C08904=1093.509,55.617,-58.520,175.678,17.080,152.502
C08905=1093.515,55.866,-58.536,175.680,17.082,152.502
C08906=1093.521,56.116,-58.551,175.682,17.083,152.502
C08907=1093.527,56.365,-58.568,175.684,17.084,152.502
C08908=1093.532,56.614,-58.583,175.686,17.085,152.502
C08909=1093.538,56.863,-58.600,175.689,17.086,152.502
C08910=1093.543,57.113,-58.617,175.690,17.087,152.501
C08911=1093.549,57.362,-58.633,175.693,17.089,152.501
C08912=1093.555,57.612,-58.648,175.695,17.090,152.501
C08913=1093.561,57.862,-58.665,175.697,17.091,152.501
C08914=1093.567,58.111,-58.681,175.699,17.092,152.501
C08915=1093.573,58.360,-58.697,175.701,17.094,152.501
C08916=1093.579,58.610,-58.713,175.703,17.094,152.500
C08917=1093.584,58.859,-58.730,175.705,17.096,152.500
C08918=1093.589,59.108,-58.746,175.708,17.097,152.500
C08919=1093.595,59.357,-58.762,175.709,17.098,152.500
C08920=1093.601,59.607,-58.779,175.712,17.100,152.500
C08921=1093.607,59.856,-58.795,175.714,17.100,152.499
C08922=1093.613,60.105,-58.811,175.716,17.102,152.499
C08923=1093.618,60.356,-58.827,175.718,17.103,152.499
C08924=1093.624,60.605,-58.844,175.720,17.104,152.499
C08925=1093.630,60.854,-58.860,175.722,17.105,152.499
C08926=1093.636,61.104,-58.876,175.725,17.107,152.499
C08927=1093.642,61.353,-58.892,175.727,17.107,152.498
C08928=1093.647,61.603,-58.909,175.728,17.108,152.498
C08929=1093.653,61.852,-58.925,175.731,17.110,152.498
C08930=1093.659,62.101,-58.942,175.733,17.110,152.498
C08931=1093.665,62.351,-58.958,175.735,17.112,152.498
C08932=1093.671,62.600,-58.974,175.737,17.113,152.497
C08933=1093.676,62.849,-58.992,175.740,17.114,152.497
C08934=1093.682,63.099,-59.008,175.742,17.115,152.497
C08935=1093.689,63.374,-59.026,175.744,17.117,152.497
C08936=1093.695,63.650,-59.044,175.747,17.118,152.497
C08937=1093.702,63.925,-59.062,175.749,17.118,152.496
C08938=1093.708,64.200,-59.080,175.751,17.120,152.496
C08939=1093.714,64.450,-59.096,175.754,17.121,152.496
C08940=1093.719,64.700,-59.113,175.755,17.122,152.496
C08941=1093.725,64.949,-59.129,175.758,17.124,152.496
C08942=1093.730,65.199,-59.146,175.760,17.125,152.495
C08943=1093.736,65.448,-59.163,175.762,17.126,152.495
C08944=1093.742,65.697,-59.180,175.764,17.127,152.495
C08945=1093.748,65.946,-59.196,175.767,17.128,152.495
C08946=1093.754,66.196,-59.213,175.769,17.129,152.495
C08947=1093.759,66.445,-59.230,175.770,17.130,152.494
C08948=1093.765,66.695,-59.246,175.773,17.131,152.494
C08949=1093.771,66.944,-59.262,175.775,17.132,152.494
C08950=1093.776,67.193,-59.280,175.777,17.134,152.494
C08951=1093.782,67.442,-59.296,175.779,17.135,152.494
C08952=1093.787,67.692,-59.313,175.782,17.136,152.493
C08953=1093.793,67.941,-59.329,175.783,17.137,152.493
C08954=1093.798,68.191,-59.346,175.786,17.138,152.493
C08955=1093.805,68.440,-59.363,175.788,17.139,152.493
C08956=1093.810,68.689,-59.380,175.790,17.141,152.493
C08957=1093.816,68.939,-59.396,175.792,17.141,152.492
C08958=1093.822,69.189,-59.413,175.795,17.143,152.492
C08959=1093.828,69.438,-59.430,175.797,17.144,152.492
C08960=1093.833,69.688,-59.447,175.799,17.145,152.492
C08961=1093.839,69.937,-59.463,175.801,17.146,152.492
C08962=1093.844,70.187,-59.480,175.804,17.147,152.491
C08963=1093.851,70.435,-59.497,175.806,17.148,152.491
C08964=1093.856,70.685,-59.514,175.808,17.149,152.491
C08965=1093.862,70.934,-59.530,175.810,17.150,152.491
C08966=1093.867,71.183,-59.548,175.812,17.152,152.491
C08967=1093.872,71.433,-59.565,175.814,17.152,152.490
C08968=1093.878,71.682,-59.581,175.817,17.154,152.490
C08969=1093.884,71.931,-59.598,175.819,17.155,152.490
C08970=1093.890,72.181,-59.615,175.821,17.156,152.490
C08971=1093.895,72.430,-59.631,175.823,17.157,152.490
C08972=1093.901,72.679,-59.649,175.826,17.158,152.489
C08973=1093.907,72.929,-59.665,175.828,17.159,152.489
C08974=1093.912,73.178,-59.683,175.830,17.161,152.489
C08975=1093.919,73.428,-59.700,175.832,17.161,152.489
C08976=1093.924,73.677,-59.716,175.835,17.163,152.488
C08977=1093.929,73.927,-59.734,175.836,17.163,152.488
C08978=1093.935,74.176,-59.750,175.839,17.165,152.488
C08979=1093.941,74.425,-59.768,175.841,17.166,152.488
C08980=1093.946,74.675,-59.785,175.844,17.167,152.488
C08981=1093.952,74.924,-59.801,175.845,17.168,152.488
C08982=1093.958,75.173,-59.818,175.848,17.169,152.487
C08983=1093.963,75.423,-59.835,175.850,17.170,152.487
C08984=1093.970,75.672,-59.853,175.852,17.171,152.487
C08985=1093.975,75.922,-59.869,175.854,17.172,152.487
C08986=1093.980,76.171,-59.887,175.857,17.173,152.486
C08987=1093.986,76.420,-59.903,175.859,17.174,152.486
C08988=1093.992,76.669,-59.921,175.861,17.176,152.486
C08989=1093.997,76.919,-59.938,175.863,17.176,152.486
C08990=1094.004,77.168,-59.955,175.866,17.177,152.485
C08991=1094.009,77.418,-59.972,175.868,17.178,152.485
C08992=1094.015,77.667,-59.989,175.870,17.179,152.485
C08993=1094.020,77.916,-60.007,175.873,17.181,152.485
C08994=1094.026,78.165,-60.023,175.875,17.182,152.485
C08995=1094.032,78.414,-60.041,175.877,17.183,152.484
C08996=1094.037,78.664,-60.058,175.879,17.183,152.484
C08997=1094.043,78.914,-60.076,175.882,17.185,152.484
C08998=1094.049,79.162,-60.093,175.884,17.186,152.484
C08999=1094.055,79.439,-60.111,175.886,17.187,152.483
C09000=1094.061,79.713,-60.131,175.889,17.188,152.483
C09001=1094.067,79.989,-60.150,175.891,17.189,152.483
C09002=1094.074,80.265,-60.168,175.894,17.190,152.483
C09003=1094.079,80.514,-60.186,175.896,17.192,152.482
C09004=1094.085,80.763,-60.203,175.898,17.192,152.482
C09005=1094.090,81.013,-60.220,175.901,17.194,152.482
C09006=1094.096,81.262,-60.238,175.903,17.194,152.482
C09007=1094.102,81.511,-60.256,175.905,17.196,152.482
C09008=1094.107,81.761,-60.273,175.907,17.197,152.481
C09009=1094.112,82.010,-60.290,175.910,17.198,152.481
C09010=1094.119,82.259,-60.307,175.912,17.199,152.481
C09011=1094.124,82.509,-60.324,175.914,17.200,152.481
C09012=1094.130,82.758,-60.342,175.917,17.201,152.480
C09013=1094.135,83.007,-60.360,175.919,17.202,152.480
C09014=1094.141,83.256,-60.377,175.921,17.203,152.480
C09015=1094.146,83.506,-60.394,175.923,17.204,152.480
C09016=1094.152,83.756,-60.412,175.926,17.205,152.479
C09017=1094.158,84.005,-60.429,175.928,17.206,152.479
C09018=1094.163,84.254,-60.447,175.931,17.207,152.479
C09019=1094.169,84.503,-60.464,175.933,17.208,152.479
C09020=1094.175,84.753,-60.482,175.935,17.209,152.478
C09021=1094.180,85.002,-60.499,175.937,17.209,152.478
C09022=1094.186,85.251,-60.517,175.940,17.211,152.478
C09023=1094.191,85.500,-60.535,175.942,17.212,152.478
C09024=1094.198,85.750,-60.552,175.944,17.213,152.477
C09025=1094.203,85.999,-60.569,175.947,17.214,152.477
C09026=1094.209,86.248,-60.586,175.949,17.215,152.477
C09027=1094.215,86.498,-60.604,175.952,17.216,152.477
C09028=1094.220,86.747,-60.622,175.953,17.217,152.476
C09029=1094.226,86.996,-60.639,175.956,17.218,152.476
C09030=1094.231,87.245,-60.657,175.958,17.219,152.476
C09031=1094.238,87.495,-60.675,175.961,17.220,152.476
C09032=1094.243,87.744,-60.692,175.963,17.220,152.475
C09033=1094.249,87.993,-60.710,175.965,17.222,152.475
C09034=1094.254,88.243,-60.727,175.968,17.223,152.475
C09035=1094.260,88.492,-60.745,175.970,17.224,152.475
C09036=1094.265,88.741,-60.762,175.973,17.225,152.474
C09037=1094.272,88.991,-60.780,175.975,17.225,152.474
C09038=1094.277,89.240,-60.798,175.977,17.227,152.474
C09039=1094.283,89.489,-60.815,175.979,17.227,152.474
C09040=1094.289,89.739,-60.833,175.982,17.228,152.473
C09041=1094.294,89.988,-60.851,175.984,17.229,152.473
C09042=1094.300,90.238,-60.869,175.987,17.230,152.473
C09043=1094.306,90.487,-60.886,175.989,17.232,152.472
C09044=1094.311,90.736,-60.904,175.991,17.232,152.472
C09045=1094.318,90.986,-60.922,175.994,17.233,152.472
C09046=1094.322,91.235,-60.940,175.996,17.234,152.472
C09047=1094.328,91.484,-60.958,175.999,17.235,152.471
C09048=1094.334,91.734,-60.976,176.000,17.236,152.471
C09049=1094.339,91.983,-60.993,176.003,17.237,152.471
C09050=1094.345,92.232,-61.011,176.006,17.238,152.470
C09051=1094.351,92.481,-61.030,176.008,17.239,152.470
C09052=1094.356,92.730,-61.047,176.011,17.240,152.470
C09053=1094.362,92.979,-61.065,176.013,17.240,152.470
C09054=1094.368,93.229,-61.083,176.015,17.242,152.469
C09055=1094.373,93.478,-61.101,176.017,17.242,152.469
C09056=1094.378,93.728,-61.119,176.020,17.243,152.469
C09057=1094.384,93.977,-61.137,176.023,17.245,152.469
C09058=1094.390,94.226,-61.154,176.025,17.245,152.468
C09059=1094.396,94.476,-61.172,176.027,17.247,152.468
C09060=1094.401,94.725,-61.191,176.029,17.247,152.468
C09061=1094.406,94.974,-61.209,176.032,17.248,152.468
C09062=1094.413,95.224,-61.227,176.034,17.249,152.467
C09063=1094.419,95.499,-61.246,176.037,17.250,152.467
C09064=1094.425,95.774,-61.267,176.040,17.251,152.467
C09065=1094.431,96.050,-61.286,176.042,17.252,152.466
C09066=1094.437,96.325,-61.306,176.045,17.253,152.466
C09067=1094.443,96.575,-61.324,176.047,17.254,152.466
C09068=1094.448,96.824,-61.343,176.050,17.255,152.465
C09069=1094.454,97.074,-61.361,176.053,17.256,152.465
C09070=1094.460,97.323,-61.378,176.054,17.257,152.465
C09071=1094.466,97.572,-61.396,176.057,17.258,152.465
C09072=1094.471,97.821,-61.415,176.059,17.259,152.464
C09073=1094.477,98.070,-61.433,176.062,17.259,152.464
C09074=1094.483,98.320,-61.451,176.064,17.260,152.464
C09075=1094.488,98.569,-61.469,176.067,17.261,152.463
C09076=1094.494,98.818,-61.487,176.069,17.262,152.463
C09077=1094.500,99.067,-61.505,176.072,17.263,152.463
C09078=1094.506,99.316,-61.524,176.074,17.264,152.463
C09079=1094.511,99.566,-61.542,176.076,17.264,152.462
C09080=1094.517,99.816,-61.560,176.079,17.266,152.462
C09081=1094.523,100.064,-61.578,176.082,17.266,152.462
C09082=1094.528,100.314,-61.596,176.084,17.267,152.461
C09083=1094.534,100.563,-61.614,176.087,17.268,152.461
C09084=1094.540,100.812,-61.633,176.088,17.269,152.461
C09085=1094.545,101.062,-61.651,176.091,17.270,152.460
C09086=1094.551,101.311,-61.670,176.094,17.271,152.460
C09087=1094.556,101.560,-61.688,176.096,17.271,152.460
